// TwinCAT 3 PLC project PLC
// ProgramVersion: 3.1.4024.0
// libraries:
//   EfficientIO Communicator, * (EfficientIO)
//   EfficientIO Energy Basic, * (EfficientIO)
//   EfficientIO ModbusTCP, * (EfficientIO)
//   Lynus Persistent Data V1, * (Lynus AG)
//   Lynus Standards, * (EfficientIO)
//   Tc2_ModbusSrv, * (Beckhoff Automation GmbH)
//   Tc2_Standard, * (Beckhoff Automation GmbH)
//   Tc2_System, * (Beckhoff Automation GmbH)
//   Tc2_Utilities, * (Beckhoff Automation GmbH)
//   Tc3_Module, * (Beckhoff Automation GmbH)
// project tree:
//   / FastTask.TcTTO, MiddleTask.TcTTO, SlowTask.TcTTO
//   FB/ FB_ModBus_100Registers_FC3.TcPOU, FB_Socomec_I31.TcPOU, FB_Socomec_IO20.TcPOU, FB_Socomec_I61.TcPOU, FB_Socomec_IO10.TcPOU
//   POUs/ MAIN.TcPOU, prgE9.TcPOU, prgComEffIO.TcPOU, prgE5.TcPOU, prgRWEffIO.TcPOU, prgVarEffIO.TcPOU
// real-time tasks:
//   TASK SlowTask: cycle T#20ms, priority 21, ADS port 351
//   TASK MiddleTask: cycle T#10ms, priority 20, ADS port 352
//   TASK FastTask: cycle T#5ms, priority 19, ADS port 353

CONFIGURATION PLC
    RESOURCE PLC ON TwinCAT3
        TASK FastTask(INTERVAL := T#5ms, PRIORITY := 19);
        TASK MiddleTask(INTERVAL := T#10ms, PRIORITY := 20);
        TASK SlowTask(INTERVAL := T#20ms, PRIORITY := 21);
        PROGRAM prgRWEffIO WITH FastTask : prgRWEffIO;
        PROGRAM prgVarEffIO WITH FastTask : prgVarEffIO;
        PROGRAM MAIN WITH MiddleTask : MAIN;
        PROGRAM prgE5 WITH MiddleTask : prgE5;
        PROGRAM prgE9 WITH MiddleTask : prgE9;
        PROGRAM prgComEffIO WITH SlowTask : prgComEffIO;
    END_RESOURCE
END_CONFIGURATION

// ---- POUs/prgRWEffIO.TcPOU
PROGRAM prgRWEffIO
VAR
	fbRW1		: FB_ReadWrite_V2;
END_VAR

fbRW1(
	eUploadType:= eSelectDataUploadType.e_Change_Intervall5min, 
	bBusy=> , 
	bError=> , 
	udiErrorCodeOut=> , 
	eErrorReadWrite_Out=> );

END_PROGRAM

// ---- POUs/prgVarEffIO.TcPOU
PROGRAM prgVarEffIO
VAR
	fbVar		: FB_VarInfo_V3;
END_VAR

fbVar(
	bReadInfo:= , 
	eTMCFile:= eSelectTMCFile.eDontUseTMCFile, 
	eSavePositionTMCFile:= eSavePositionOnPLC.ePostionC, 
	udiCounterFoundVariables=> , 
	bError=> , 
	bBusy=> , 
	byProgress=> , 
	udiErrorCodeOut=> , 
	eErrorVarInfo_Out=> , 
	sVarWithError=> );

END_PROGRAM

// ---- POUs/MAIN.TcPOU
PROGRAM MAIN
VAR
	FB_Read_MB :FB_ModBus_100Registers_FC3;
	m_Enable: BOOL ;
	str_IP: STRING(15):= '192.168.8.2';
	word_Adress: WORD;
	usint_Quantity: USINT;
	byte_slaveID: BYTE;

	lr_Mischanlage_Gesamt_Freq : LREAL;		//{#lynus.ag#()}
	lr_Mischanlage_Gesamt_L1N : LREAL;		//{#lynus.ag#()}
	lr_Mischanlage_Gesamt_L2N : LREAL;		//{#lynus.ag#()}
	lr_Mischanlage_Gesamt_L3N : LREAL;		//{#lynus.ag#()}
	lr_Mischanlage_Gesamt_L1L2 : LREAL;		//{#lynus.ag#()}
	lr_Mischanlage_Gesamt_L2L3 : LREAL;		//{#lynus.ag#()}
	lr_Mischanlage_Gesamt_L3L1 : LREAL;		//{#lynus.ag#()}
	lr_Mischanlage_Gesamt_I1 : LREAL;		//{#lynus.ag#()}
	lr_Mischanlage_Gesamt_I2 : LREAL;		//{#lynus.ag#()}
	lr_Mischanlage_Gesamt_I3 : LREAL;		//{#lynus.ag#()}
	lr_Mischanlage_Gesamt_N : LREAL;		//{#lynus.ag#()}
	lr_Mischanlage_Gesamt_S : LREAL;		//{#lynus.ag#()}
	lr_Mischanlage_Gesamt_P : LREAL;		//{#lynus.ag#()}
	lr_Mischanlage_Gesamt_Q : LREAL;		//{#lynus.ag#()}
	lr_Mischanlage_Gesamt_PF : LREAL;		//{#lynus.ag#()}
	
	lr_VerteilerRC_Kalt_Freq : LREAL;		//{#lynus.ag#()}
	lr_VerteilerRC_Kalt_L1N : LREAL;		//{#lynus.ag#()}
	lr_VerteilerRC_Kalt_L2N : LREAL;		//{#lynus.ag#()}
	lr_VerteilerRC_Kalt_L3N : LREAL;		//{#lynus.ag#()}
	lr_VerteilerRC_Kalt_L1L2 : LREAL;		//{#lynus.ag#()}
	lr_VerteilerRC_Kalt_L2L3 : LREAL;		//{#lynus.ag#()}
	lr_VerteilerRC_Kalt_L3L1 : LREAL;		//{#lynus.ag#()}
	lr_VerteilerRC_Kalt_I1 : LREAL;			//{#lynus.ag#()}
	lr_VerteilerRC_Kalt_I2 : LREAL;			//{#lynus.ag#()}
	lr_VerteilerRC_Kalt_I3 : LREAL;			//{#lynus.ag#()}
	lr_VerteilerRC_Kalt_N : LREAL;			//{#lynus.ag#()}
	lr_VerteilerRC_Kalt_S : LREAL;			//{#lynus.ag#()}
	lr_VerteilerRC_Kalt_P : LREAL;			//{#lynus.ag#()}
	lr_VerteilerRC_Kalt_Q : LREAL;			//{#lynus.ag#()}
	lr_VerteilerRC_Kalt_PF : LREAL;			//{#lynus.ag#()}
	

	lr_Begleitheizung_Freq : LREAL;			//{#lynus.ag#()}
	lr_Begleitheizung_L1N : LREAL;			//{#lynus.ag#()}
	lr_Begleitheizung_L2N : LREAL;			//{#lynus.ag#()}
	lr_Begleitheizung_L3N : LREAL;			//{#lynus.ag#()}
	lr_Begleitheizung_L1L2 : LREAL;			//{#lynus.ag#()}
	lr_Begleitheizung_L2L3 : LREAL;			//{#lynus.ag#()}
	lr_Begleitheizung_L3L1 : LREAL;			//{#lynus.ag#()}
	lr_Begleitheizung_I1 : LREAL;			//{#lynus.ag#()}
	lr_Begleitheizung_I2 : LREAL;			//{#lynus.ag#()}
	lr_Begleitheizung_I3 : LREAL;			//{#lynus.ag#()}
	lr_Begleitheizung_N : LREAL;			//{#lynus.ag#()}
	lr_Begleitheizung_S : LREAL;			//{#lynus.ag#()}
	lr_Begleitheizung_P : LREAL;			//{#lynus.ag#()}
	lr_Begleitheizung_Q : LREAL;			//{#lynus.ag#()}
	lr_Begleitheizung_PF : LREAL;			//{#lynus.ag#()}

	lr_Nebenantriebe_Freq : LREAL;			//{#lynus.ag#()}
	lr_Nebenantriebe_L1N : LREAL;			//{#lynus.ag#()}
	lr_Nebenantriebe_L2N : LREAL;			//{#lynus.ag#()}
	lr_Nebenantriebe_L3N : LREAL;			//{#lynus.ag#()}
	lr_Nebenantriebe_L1L2 : LREAL;			//{#lynus.ag#()}
	lr_Nebenantriebe_L2L3 : LREAL;			//{#lynus.ag#()}
	lr_Nebenantriebe_L3L1 : LREAL;			//{#lynus.ag#()}
	lr_Nebenantriebe_I1 : LREAL;			//{#lynus.ag#()}
	lr_Nebenantriebe_I2 : LREAL;			//{#lynus.ag#()}
	lr_Nebenantriebe_I3 : LREAL;			//{#lynus.ag#()}
	lr_Nebenantriebe_N : LREAL;				//{#lynus.ag#()}
	lr_Nebenantriebe_S : LREAL;				//{#lynus.ag#()}
	lr_Nebenantriebe_P : LREAL;				//{#lynus.ag#()}
	lr_Nebenantriebe_Q : LREAL;				//{#lynus.ag#()}
	lr_Nebenantriebe_PF : LREAL;			//{#lynus.ag#()}
	
	lr_Rest_P : LREAL;								//{#lynus.ag#()}
	lr_GasmessungWTMenge_m3h 	: LREAL;			//{#lynus.ag#()}
	lr_GasmessungWTMenge_m3h_2 	: LREAL;			//{#lynus.ag#()}
	lr_GasmessungWTTemp_C 		: LREAL;			//{#lynus.ag#()}
	lr_GasmessungWTDruck_bar 	: LREAL;			//{#lynus.ag#()}
	m_Brennerstart			 	: BOOL;			//{#lynus.ag#()}
	m_Mischerstart			 	: BOOL;			//{#lynus.ag#()}
	m_Oelzaehler			 	: BOOL;			//{#lynus.ag#()}
	
	FB_Read_Socomec_I61 	: FB_Socomec_I61;
	FB_Read_Socomec_IO20	: FB_Socomec_IO20;
	FB_Read_Socomec_IO10	: FB_Socomec_IO10;
	i_State_ModbusCall: INT;				
	ton_TimeOutState: ton;
	tof_TimeOut_Active: tof;
	i_State_ModbusCall_old: INT;
	int_errorCount: INT;
	m_TimeOutActive: BOOL;					//{#lynus.ag#()}
	i_State_ErrorActive: INT;				//{#lynus.ag#()}
	lr_Rest_P_Temp: LREAL;
END_VAR


lr_Rest_P := LIMIT(	0,
					lr_Mischanlage_Gesamt_P - lr_VerteilerRC_Kalt_P - lr_Begleitheizung_P - lr_Nebenantriebe_P
						- prgE5.lr_RC_Anlage_P - prgE5.lr_RC_Trommel_P  
						- prgE9.lr_Bitumentank_4_P - prgE9.lr_Dosierpumpe_1_P - prgE9.lr_Bitumenfuellpumpe_1_P - prgE9.lr_Dosierpumpe_2_P  - prgE9.lr_Bitumentank_1_P - prgE9.lr_Bitumentank_2_P - prgE9.lr_Bitumentank_3_P
					,1000);
lr_Rest_P_Temp :=	lr_Mischanlage_Gesamt_P - lr_VerteilerRC_Kalt_P - lr_Begleitheizung_P - lr_Nebenantriebe_P
						- prgE5.lr_RC_Anlage_P - prgE5.lr_RC_Trommel_P  
						- prgE9.lr_Bitumentank_4_P - prgE9.lr_Dosierpumpe_1_P - prgE9.lr_Bitumenfuellpumpe_1_P - prgE9.lr_Dosierpumpe_2_P  - prgE9.lr_Bitumentank_1_P - prgE9.lr_Bitumentank_2_P - prgE9.lr_Bitumentank_3_P;
CASE i_State_ModbusCall OF
	0: 	// wait state
		i_State_ModbusCall := 10;
	
	10:	// first Modbus Poll Call
		FB_Read_Socomec_I61.m_Start := TRUE;
		FB_Read_Socomec_I61.byte_slaveID := 3;
		FB_Read_Socomec_I61.w_Adress := 18442;
		i_State_ModbusCall := i_State_ModbusCall + 1;
	
	11: // wait for received data
		FB_Read_Socomec_I61.m_Start := FALSE;
		IF FB_Read_Socomec_I61.iStateModbusRead = 30 THEN
			lr_Mischanlage_Gesamt_Freq	:=		FB_Read_Socomec_I61.lr_Freq_Hz	;	
			lr_Mischanlage_Gesamt_L1N	:=		FB_Read_Socomec_I61.lr_L1N_V	;	
			lr_Mischanlage_Gesamt_L2N	:=		FB_Read_Socomec_I61.lr_L2N_V	;	
			lr_Mischanlage_Gesamt_L3N	:=		FB_Read_Socomec_I61.lr_L3N_V	;	
			lr_Mischanlage_Gesamt_L1L2	:=		FB_Read_Socomec_I61.lr_L1L2_V	;	
			lr_Mischanlage_Gesamt_L2L3	:=		FB_Read_Socomec_I61.lr_L2L3_V	;	
			lr_Mischanlage_Gesamt_L3L1	:=		FB_Read_Socomec_I61.lr_L3L1_V	;	
			lr_Mischanlage_Gesamt_I1	:=		FB_Read_Socomec_I61.lr_I1_A		;	
			lr_Mischanlage_Gesamt_I2	:=		FB_Read_Socomec_I61.lr_I2_A		;	
			lr_Mischanlage_Gesamt_I3	:=		FB_Read_Socomec_I61.lr_I3_A		;	
			lr_Mischanlage_Gesamt_N		:=		FB_Read_Socomec_I61.lr_N_A		;	
			lr_Mischanlage_Gesamt_P		:=		FB_Read_Socomec_I61.lr_P_kW		;	
			lr_Mischanlage_Gesamt_Q		:=		FB_Read_Socomec_I61.lr_Q_kVAr	;	
			lr_Mischanlage_Gesamt_S		:=		FB_Read_Socomec_I61.lr_S_kVA	;	
			lr_Mischanlage_Gesamt_PF	:=		FB_Read_Socomec_I61.lr_PF		;		
			
			i_State_ModbusCall := i_State_ModbusCall +1;
		END_IF            
		IF FB_Read_Socomec_I61.iStateModbusError = 300 OR ton_TimeOutState.Q THEN
			i_State_ModbusCall := i_State_ModbusCall +1;
		END_IF
	
	12: // wait for FB_Read_Socomec_I61 to be in state 0
		IF FB_Read_Socomec_I61.iStateModbusRead = 0 OR ton_TimeOutState.Q THEN
			i_State_ModbusCall := i_State_ModbusCall + 8;
		END_IF

	20:	// next Modbus Poll Call
		FB_Read_Socomec_I61.m_Start := TRUE;
		FB_Read_Socomec_I61.byte_slaveID := 4;
		FB_Read_Socomec_I61.w_Adress := 18442;
		i_State_ModbusCall := i_State_ModbusCall + 1;
	
	21: // wait for received data
		FB_Read_Socomec_I61.m_Start := FALSE;
		IF FB_Read_Socomec_I61.iStateModbusRead = 30 THEN
			lr_VerteilerRC_Kalt_Freq	:=		FB_Read_Socomec_I61.lr_Freq_Hz	;	
			lr_VerteilerRC_Kalt_L1N		:=		FB_Read_Socomec_I61.lr_L1N_V	;	
			lr_VerteilerRC_Kalt_L2N		:=		FB_Read_Socomec_I61.lr_L2N_V	;	
			lr_VerteilerRC_Kalt_L3N		:=		FB_Read_Socomec_I61.lr_L3N_V	;	
			lr_VerteilerRC_Kalt_L1L2	:=		FB_Read_Socomec_I61.lr_L1L2_V	;	
			lr_VerteilerRC_Kalt_L2L3	:=		FB_Read_Socomec_I61.lr_L2L3_V	;	
			lr_VerteilerRC_Kalt_L3L1	:=		FB_Read_Socomec_I61.lr_L3L1_V	;	
			lr_VerteilerRC_Kalt_I1		:=		FB_Read_Socomec_I61.lr_I1_A		;	
			lr_VerteilerRC_Kalt_I2		:=		FB_Read_Socomec_I61.lr_I2_A		;	
			lr_VerteilerRC_Kalt_I3		:=		FB_Read_Socomec_I61.lr_I3_A		;	
			lr_VerteilerRC_Kalt_N		:=		FB_Read_Socomec_I61.lr_N_A		;	
			lr_VerteilerRC_Kalt_P		:=		FB_Read_Socomec_I61.lr_P_kW		;	
			lr_VerteilerRC_Kalt_Q		:=		FB_Read_Socomec_I61.lr_Q_kVAr	;	
			lr_VerteilerRC_Kalt_S		:=		FB_Read_Socomec_I61.lr_S_kVA	;	
			lr_VerteilerRC_Kalt_PF		:=		FB_Read_Socomec_I61.lr_PF		;		
			
			i_State_ModbusCall := i_State_ModbusCall +1;
		END_IF            
		IF FB_Read_Socomec_I61.iStateModbusError = 300 OR ton_TimeOutState.Q THEN
			i_State_ModbusCall := i_State_ModbusCall +1;
		END_IF
	
	22: // wait for FB_Read_Socomec_I61 to be in state 0
		IF FB_Read_Socomec_I61.iStateModbusRead = 0 OR ton_TimeOutState.Q THEN
			i_State_ModbusCall := i_State_ModbusCall + 8;
		END_IF
	
	30:	// next Modbus Poll Call
		FB_Read_Socomec_I61.m_Start := TRUE;
		FB_Read_Socomec_I61.byte_slaveID := 3;
		FB_Read_Socomec_I61.w_Adress := 20490;
		i_State_ModbusCall := i_State_ModbusCall + 1;
	
	31: // wait for received data
		FB_Read_Socomec_I61.m_Start := FALSE;
		IF FB_Read_Socomec_I61.iStateModbusRead = 30 THEN
			lr_Begleitheizung_Freq	:=		FB_Read_Socomec_I61.lr_Freq_Hz	;	
			lr_Begleitheizung_L1N	:=		FB_Read_Socomec_I61.lr_L1N_V	;	
			lr_Begleitheizung_L2N	:=		FB_Read_Socomec_I61.lr_L2N_V	;	
			lr_Begleitheizung_L3N	:=		FB_Read_Socomec_I61.lr_L3N_V	;	
			lr_Begleitheizung_L1L2	:=		FB_Read_Socomec_I61.lr_L1L2_V	;	
			lr_Begleitheizung_L2L3	:=		FB_Read_Socomec_I61.lr_L2L3_V	;	
			lr_Begleitheizung_L3L1	:=		FB_Read_Socomec_I61.lr_L3L1_V	;	
			lr_Begleitheizung_I1	:=		FB_Read_Socomec_I61.lr_I1_A		;	
			lr_Begleitheizung_I2	:=		FB_Read_Socomec_I61.lr_I2_A		;	
			lr_Begleitheizung_I3	:=		FB_Read_Socomec_I61.lr_I3_A		;	
			lr_Begleitheizung_N		:=		FB_Read_Socomec_I61.lr_N_A		;	
			lr_Begleitheizung_P		:=		FB_Read_Socomec_I61.lr_P_kW		;	
			lr_Begleitheizung_Q		:=		FB_Read_Socomec_I61.lr_Q_kVAr	;	
			lr_Begleitheizung_S		:=		FB_Read_Socomec_I61.lr_S_kVA	;	
			lr_Begleitheizung_PF	:=		FB_Read_Socomec_I61.lr_PF		;		
			
			i_State_ModbusCall := i_State_ModbusCall +1;
		END_IF            
		IF FB_Read_Socomec_I61.iStateModbusError = 300 OR ton_TimeOutState.Q THEN
			i_State_ModbusCall := i_State_ModbusCall +1;
		END_IF
	
	32: // wait for FB_Read_Socomec_I61 to be in state 0
		IF FB_Read_Socomec_I61.iStateModbusRead = 0 OR ton_TimeOutState.Q THEN
			i_State_ModbusCall := i_State_ModbusCall + 8;
		END_IF
	
	40:	// next Modbus Poll Call
		FB_Read_Socomec_I61.m_Start := TRUE;
		FB_Read_Socomec_I61.byte_slaveID := 4;
		FB_Read_Socomec_I61.w_Adress := 20490;
		i_State_ModbusCall := i_State_ModbusCall + 1;
	
	41: // wait for received data
		FB_Read_Socomec_I61.m_Start := FALSE;
		IF FB_Read_Socomec_I61.iStateModbusRead = 30 THEN
			lr_Nebenantriebe_Freq	:=		FB_Read_Socomec_I61.lr_Freq_Hz	;	
			lr_Nebenantriebe_L1N	:=		FB_Read_Socomec_I61.lr_L1N_V	;	
			lr_Nebenantriebe_L2N	:=		FB_Read_Socomec_I61.lr_L2N_V	;	
			lr_Nebenantriebe_L3N	:=		FB_Read_Socomec_I61.lr_L3N_V	;	
			lr_Nebenantriebe_L1L2	:=		FB_Read_Socomec_I61.lr_L1L2_V	;	
			lr_Nebenantriebe_L2L3	:=		FB_Read_Socomec_I61.lr_L2L3_V	;	
			lr_Nebenantriebe_L3L1	:=		FB_Read_Socomec_I61.lr_L3L1_V	;	
			lr_Nebenantriebe_I1		:=		FB_Read_Socomec_I61.lr_I1_A		;	
			lr_Nebenantriebe_I2		:=		FB_Read_Socomec_I61.lr_I2_A		;	
			lr_Nebenantriebe_I3		:=		FB_Read_Socomec_I61.lr_I3_A		;	
			lr_Nebenantriebe_N		:=		FB_Read_Socomec_I61.lr_N_A		;	
			lr_Nebenantriebe_P		:=		FB_Read_Socomec_I61.lr_P_kW		;	
			lr_Nebenantriebe_Q		:=		FB_Read_Socomec_I61.lr_Q_kVAr	;	
			lr_Nebenantriebe_S		:=		FB_Read_Socomec_I61.lr_S_kVA	;	
			lr_Nebenantriebe_PF		:=		FB_Read_Socomec_I61.lr_PF		;		
			
			i_State_ModbusCall := i_State_ModbusCall +1;
		END_IF            
		IF FB_Read_Socomec_I61.iStateModbusError = 300 OR ton_TimeOutState.Q THEN
			i_State_ModbusCall := i_State_ModbusCall +1;
		END_IF
	
	42: // wait for FB_Read_Socomec_I61 to be in state 0
		IF FB_Read_Socomec_I61.iStateModbusRead = 0 OR ton_TimeOutState.Q THEN
			i_State_ModbusCall := i_State_ModbusCall + 8;
		END_IF


	50:	// next Modbus Poll Call		first IO20 call
		FB_Read_Socomec_IO20.m_Start := TRUE;
		FB_Read_Socomec_IO20.byte_slaveID := 5;
		FB_Read_Socomec_IO20.w_Adress := 11589;
		i_State_ModbusCall := i_State_ModbusCall + 1;
	
	51: // wait for received data
		FB_Read_Socomec_IO20.m_Start := FALSE;
		IF FB_Read_Socomec_IO20.iStateModbusRead = 30 THEN
			lr_GasmessungWTMenge_m3h := LIMIT(0,2150.0/16.0*(FB_Read_Socomec_IO20.lr_Value_mA-4),2150);		// 4-20mA = 0-2150 m3/h
			lr_GasmessungWTMenge_m3h_2 := LIMIT(0,FB_Read_Socomec_IO20.lr_Value_mA,2150);					// plain Output Socomec
			i_State_ModbusCall := i_State_ModbusCall +1;
		END_IF            
		IF FB_Read_Socomec_I61.iStateModbusError = 300 OR ton_TimeOutState.Q THEN
			i_State_ModbusCall := i_State_ModbusCall +1;
		END_IF
	
	52: // wait for FB_Read_Socomec_IO20 to be in state 0
		IF FB_Read_Socomec_IO20.iStateModbusRead = 0 OR ton_TimeOutState.Q THEN
			i_State_ModbusCall := i_State_ModbusCall + 8;
		END_IF
		
	60:	// next Modbus Poll Call		second IO20 call
		FB_Read_Socomec_IO20.m_Start := TRUE;
		FB_Read_Socomec_IO20.byte_slaveID := 5;
		FB_Read_Socomec_IO20.w_Adress := 11621;
		i_State_ModbusCall := i_State_ModbusCall + 1;
	
	61: // wait for received data
		FB_Read_Socomec_IO20.m_Start := FALSE;
		IF FB_Read_Socomec_IO20.iStateModbusRead = 30 THEN
			lr_GasmessungWTTemp_C := LIMIT(-20,100.0/16.0*(FB_Read_Socomec_IO20.lr_Value_mA-4)-20,80);		// 4-20mA = -20-80 °C
				
			i_State_ModbusCall := i_State_ModbusCall +1;
		END_IF            
		IF FB_Read_Socomec_IO20.iStateModbusError = 300 OR ton_TimeOutState.Q THEN
			i_State_ModbusCall := i_State_ModbusCall +1;
		END_IF
	
	62: // wait for FB_Read_Socomec_IO20 to be in state 0
		IF FB_Read_Socomec_IO20.iStateModbusRead = 0 OR ton_TimeOutState.Q THEN
			i_State_ModbusCall := i_State_ModbusCall + 8;
		END_IF
	70:	// next Modbus Poll Call		third IO20 call
		FB_Read_Socomec_IO20.m_Start := TRUE;
		FB_Read_Socomec_IO20.byte_slaveID := 6;
		FB_Read_Socomec_IO20.w_Adress := 11589;
		i_State_ModbusCall := i_State_ModbusCall + 1;
	
	71: // wait for received data
		FB_Read_Socomec_IO20.m_Start := FALSE;
		IF FB_Read_Socomec_IO20.iStateModbusRead = 30 THEN
			lr_GasmessungWTDruck_bar :=	LIMIT(0,(5.0/16.0) * (FB_Read_Socomec_IO20.lr_Value_mA-4),5);		// 4-20mA = 0-5 bar
			i_State_ModbusCall := i_State_ModbusCall +1;
		END_IF            
		IF FB_Read_Socomec_IO20.iStateModbusError = 300 OR ton_TimeOutState.Q THEN
			i_State_ModbusCall := i_State_ModbusCall +1;
		END_IF
	
	72: // wait for FB_Read_Socomec_IO20 to be in state 0
		IF FB_Read_Socomec_IO20.iStateModbusRead = 0 OR ton_TimeOutState.Q THEN
			i_State_ModbusCall := i_State_ModbusCall + 8;
		END_IF

	80:	// next Modbus Poll Call		first IO20 call
		FB_Read_Socomec_IO10.m_Start := TRUE;
		FB_Read_Socomec_IO10.byte_slaveID := 7;
		FB_Read_Socomec_IO10.w_Adress := 11520;
		i_State_ModbusCall := i_State_ModbusCall + 1;
	
	81: // wait for received data
		FB_Read_Socomec_IO10.m_Start := FALSE;
		IF FB_Read_Socomec_IO10.iStateModbusRead = 30 THEN
			m_Brennerstart := FB_Read_Socomec_IO10.m_Input_Active;		
				
			i_State_ModbusCall := i_State_ModbusCall +1;
		END_IF            
		IF FB_Read_Socomec_IO10.iStateModbusError = 300 OR ton_TimeOutState.Q THEN
			i_State_ModbusCall := i_State_ModbusCall +1;
		END_IF
	
	82: // wait for FB_Read_Socomec_IO10 to be in state 0
		IF FB_Read_Socomec_IO10.iStateModbusRead = 0 OR ton_TimeOutState.Q THEN
			i_State_ModbusCall := i_State_ModbusCall + 8;
		END_IF

	90:	// next Modbus Poll Call		first IO20 call
		FB_Read_Socomec_IO10.m_Start := TRUE;
		FB_Read_Socomec_IO10.byte_slaveID := 7;
		FB_Read_Socomec_IO10.w_Adress := 11522;
		i_State_ModbusCall := i_State_ModbusCall + 1;
	
	91: // wait for received data
		FB_Read_Socomec_IO10.m_Start := FALSE;
		IF FB_Read_Socomec_IO10.iStateModbusRead = 30 THEN
			m_Mischerstart := FB_Read_Socomec_IO10.m_Input_Active;		
				
			i_State_ModbusCall := i_State_ModbusCall +1;
		END_IF            
		IF FB_Read_Socomec_IO10.iStateModbusError = 300 OR ton_TimeOutState.Q THEN
			i_State_ModbusCall := i_State_ModbusCall +1;
		END_IF
	
	92: // wait for FB_Read_Socomec_IO10 to be in state 0
		IF FB_Read_Socomec_IO10.iStateModbusRead = 0 OR ton_TimeOutState.Q THEN
			i_State_ModbusCall := i_State_ModbusCall + 8;
		END_IF
	100:	// next Modbus Poll Call		first IO20 call
		FB_Read_Socomec_IO10.m_Start := TRUE;
		FB_Read_Socomec_IO10.byte_slaveID := 7;
		FB_Read_Socomec_IO10.w_Adress := 11524;
		i_State_ModbusCall := i_State_ModbusCall + 1;
	
	101: // wait for received data
		FB_Read_Socomec_IO10.m_Start := FALSE;
		IF FB_Read_Socomec_IO10.iStateModbusRead = 30 THEN
			m_Oelzaehler := FB_Read_Socomec_IO10.m_Input_Active;		
				
			i_State_ModbusCall := i_State_ModbusCall +1;
		END_IF            
		IF FB_Read_Socomec_IO10.iStateModbusError = 300 OR ton_TimeOutState.Q THEN
			i_State_ModbusCall := i_State_ModbusCall +1;
		END_IF
	
	102: // wait for FB_Read_Socomec_IO10 to be in state 0
		IF FB_Read_Socomec_IO10.iStateModbusRead = 0 OR ton_TimeOutState.Q THEN
			i_State_ModbusCall := i_State_ModbusCall + 8;
		END_IF				
		
	110: 
		i_State_ModbusCall := 0;
END_CASE

ton_TimeOutState(	IN:= i_State_ModbusCall = i_State_ModbusCall_old, 
					PT:= T#30S, 
					Q=> , 
					ET=> );

i_State_ModbusCall_old := i_State_ModbusCall; 

IF ton_TimeOutState.Q THEN
//	i_State_ModbusCall := 0;
	int_errorCount := int_errorCount  + 1; 
END_IF


tof_TimeOut_Active(	IN:= ton_TimeOutState.Q, 
					PT:=	T#5S , 
					Q=> m_TimeOutActive, 
					ET=> );
IF tof_TimeOut_Active.Q THEN
	 i_State_ErrorActive := i_State_ModbusCall; 
END_IF


FB_Read_Socomec_I61(
	m_Start:= , 
	str_IPAdress:= str_IP , 
	w_Adress:= , 
	uint_port:= , 
	byte_slaveID:= , 
	m_PollSuccessful=> , 
	lr_Freq_Hz=> , 
	lr_L1N_V=> , 
	lr_L2N_V=> , 
	lr_L3N_V=> , 
	lr_L1L2_V=> , 
	lr_L2L3_V=> , 
	lr_L3L1_V=> , 
	lr_I1_A=> , 
	lr_I2_A=> , 
	lr_I3_A=> , 
	lr_N_A=> , 
	lr_P_kW=> , 
	lr_Q_kVAr=> , 
	lr_S_kVA=> , 
	lr_PF=> , 
	udint_Error_ID=> );

FB_Read_Socomec_IO20(
	m_Start:= , 
	str_IPAdress:= str_IP, 
	w_Adress:= , 
	uint_port:= , 
	byte_slaveID:= , 
	m_PollSuccessful=> , 
	lr_Value_mA=> , 
	udint_Error_ID=> );

FB_Read_Socomec_IO10(
	m_Start:= , 
	str_IPAdress:= str_IP , 
	w_Adress:= , 
	uint_port:= , 
	byte_slaveID:= , 
	m_PollSuccessful=> , 
	m_Input_Active=> , 
	udint_Error_ID=> );	


FB_Read_MB(
	m_Enable:= m_Enable, 
	str_IPAdress:= str_IP,
	w_Adress:= word_Adress, 
	usint_Quantity:= usint_Quantity, 
	byte_slaveID:=byte_slaveID,
	uint_port := ,
	m_PollSuccessful=> , 
	w_Array_Received=> , 
	udint_Error_ID=> );

END_PROGRAM

// ---- FB/FB_ModBus_100Registers_FC3.TcPOU
FUNCTION_BLOCK FB_ModBus_100Registers_FC3
VAR_INPUT PERSISTENT
	m_Enable					: BOOL;						//Enable the Fuctionblock and his logic
	str_IPAdress				: STRING(15);				//IP Adress of the meter
	w_Adress					: WORD;						//modbus adress
	usint_Quantity				: USINT;					//Number of Words to get polled, max 100
	uint_port					: UINT:=502;				//ModbusPort
	byte_slaveID				: BYTE;						//SlaveID of the meter
END_VAR
VAR_OUTPUT
	m_PollSuccessful			: BOOL;						//Poll succesfull		
	w_Array_Received			: ARRAY[1..100] OF WORD;	// received data
	udint_Error_ID				: UDINT;					// ERR ID FB_MBReadRegs
END_VAR
VAR
	
	timer_Delay					: TON;						//Timer for Delay between Requests
	
	timer_DelayStart			: TON;						//Timer to start the state machine with Delay after enabling or after the system ist restartet
	
	timer_TimeOut				: TON;						//Timer for Timeout MB Read
	
	iStateModbusRead			: INT;						//State machine for read out Data over Modbus RTU
	
	fbMBRead_FC3				: FB_MBReadRegs  ;		//Modbus Read Function (FC3)
	
	ftrig_PEnable				: f_trig;					//Internal positive Edge
	
	iStateModbusError			: INT;						//State machine for error out Data over Modbus TCP/IP	
	
	FPError_FC_3				: R_TRIG;					//Internal positive Edge
	
	arrBuffer_FC3				: ARRAY[1..100] OF WORD;		//Buffer with Data from FC3
	
	timer_Connection_ok			: TON;
	int_Data_Received			: INT;
	
	m_MBTCPError				: BOOL;
	
	int_Data_Received_old		: INT;
	
	timer_Connection_ok_TOF	: TOF;
	
	fbConvertWordToDword		: FB_CV_WORD_TO_DWORD;			//Convert Word to Dword
	
	m_Poll_ok: BOOL;
	
	timer_Wait: Ton;
	int_TimeoutError: INT;
	int_FC3Error: INT;

END_VAR

(*	{attribute 'hide'}--------------------------------------------------------------------------------------------Limits-------------------------------------------------------------------------------------*)

w_Adress := LIMIT(0,w_Adress,60000);
usint_Quantity := LIMIT(1,usint_Quantity,100);
	
(*--------------------------------------------------------------------------------------------State Machine Read--------------------------------------------------------------------------------------*)

//Timer for Delay
timer_Delay(IN:= , PT:= T#50MS, Q=> , ET=> );

//Timeout Timer is dissabled when the Init Step is aktiv or the function is not enabled
IF iStateModbusRead = 0 OR NOT m_Enable THEN 
	timer_Timeout.IN := FALSE; 
END_IF
timer_Timeout(IN:= , PT:= T#1S, Q=> , ET=> );

//Enable with Delay that not all sockets have to be created at the same time
timer_DelayStart(IN:= m_Enable, PT:= T#1S, Q=> , ET=> );
ftrig_PEnable(CLK:= timer_DelayStart.Q, Q=> );

IF ftrig_PEnable.Q AND iStateModbusRead = 0 THEN 
	iStateModbusRead := 1; 
END_IF		
		
//Not Enabled
IF NOT m_Enable THEN 
	iStateModbusRead := 0; 
	iStateModbusError := 0; 
END_IF		
		
CASE iStateModbusRead OF

	0://Init Step 
		timer_Delay.IN := FALSE;
		fbMBRead_FC3.bExecute := FALSE;
		m_Poll_ok:=FALSE;
		int_Data_Received:=0;
	
		iStateModbusRead := 1;
	
	1://read the required registers
		//Start Read
		fbMBRead_FC3.nQuantity := usint_Quantity;
		fbMBRead_FC3.nMBAddr := w_Adress;
		fbMBRead_FC3.bExecute := TRUE;
		fbMBRead_FC3.nUnitID := byte_slaveID;
		timer_Timeout.IN := TRUE;
		IF fbMBRead_FC3.bBusy THEN 
			timer_Delay.IN := TRUE; 
		END_IF
		
		//Wait for Delay, copy Data and then next step
		IF NOT fbMBRead_FC3.bBusy AND NOT fbMBRead_FC3.bError AND timer_Delay.Q THEN
			m_Poll_ok:=TRUE;
			int_Data_Received:=int_Data_Received+1;
			m_MBTCPError := FALSE; 
			
			w_Array_Received := arrBuffer_FC3;
			
			
			//Go to Next Step
			timer_Timeout.IN := FALSE;
			fbMBRead_FC3.bExecute := FALSE;
			timer_Delay.IN := FALSE;		
			iStateModbusRead := 3;
		END_IF	

		//Error or Timeout
		IF FPError_FC_3.Q THEN 
			iStateModbusError := 300;
			int_FC3Error := int_FC3Error+1;
		ELSIF timer_Timeout.Q THEN  
			timer_Timeout.IN := FALSE; 	
			iStateModbusError := 300;
			int_TimeoutError := int_TimeoutError+1;
		END_IF
		
	
	3://Wait and go to step 1
		//1 because 0 is the Init Step for Read
		timer_Wait.IN := TRUE;
		
		IF timer_Wait.Q = TRUE THEN
			iStateModbusRead := 1;
			timer_Wait.IN :=FALSE;
		END_IF

			
		
		//Error on Master, changes on Inputs or Timeout
		IF timer_Timeout.Q THEN 
			iStateModbusError := 300; 
		END_IF
	
END_CASE

(* wait timer*)

timer_Wait(PT:=T#3S);


(*------------------------------------------------------------------Error and Warning----------------------------------------------------------------------------*)	
 
timer_Connection_ok			(In:=int_Data_Received<>int_Data_Received_old,PT:=T#10S);
timer_Connection_ok_TOF		(In:=NOT(int_Data_Received<>int_Data_Received_old) AND int_Data_Received>3 ,PT:=T#20S);
int_Data_Received_old:=int_Data_Received;
m_PollSuccessful:=NOT timer_Connection_ok.Q AND timer_Connection_ok_TOF.Q ;

(*------------------------------------------------------------------------------------------Modbus TCP Functions---------------------------------------------------------------------------------------------*)

fbMBRead_FC3(	sIPAddr:= str_IPAdress, 
				nTCPPort:= uint_port,
				cbLength:= SIZEOF(arrBuffer_FC3), 
				pDestAddr:= ADR(arrBuffer_FC3), 
				tTimeout:= T#10S,
				nErrId => udint_Error_ID);

FPError_FC_3(CLK:= fbMBRead_FC3.bError, Q=> );		

(*------------------------------------------------------------------------------------------State Machine Error---------------------------------------------------------------------------------------------*)	

CASE iStateModbusError OF
	
	300://Error
		timer_Wait.IN :=TRUE;
		timer_Delay.IN := FALSE;
		fbMBRead_FC3.bExecute := FALSE;
		m_MBTCPError := TRUE; 		
		m_Poll_ok:=FALSE;
		int_Data_Received:=0;
				//Restart from new with the Read out part after an Error
		IF timer_Wait.Q = TRUE THEN
			iStateModbusRead := 0;	
			iStateModbusError := 0;
			timer_Wait.IN :=FALSE;
			timer_Timeout.IN := FALSE;
		END_IF		
							
END_CASE

END_FUNCTION_BLOCK

// ---- FB/FB_Socomec_I61.TcPOU
FUNCTION_BLOCK FB_Socomec_I61
VAR_INPUT PERSISTENT
	m_Start						: BOOL;						//starts one modbus read out
	str_IPAdress				: STRING(15);				//IP Adress of the meter
	w_Adress					: WORD;						//modbus adress
	uint_port					: UINT:=502;				//ModbusPort
	byte_slaveID				: BYTE;						//SlaveID of the meter
END_VAR
VAR_OUTPUT
	m_PollSuccessful			: BOOL;						//Poll succesfull		
	lr_Freq_Hz					: LREAL;
	lr_L1N_V					: LREAL;	
	lr_L2N_V					: LREAL;	
	lr_L3N_V					: LREAL;	
	lr_L1L2_V					: LREAL;	
	lr_L2L3_V					: LREAL;	
	lr_L3L1_V					: LREAL;	
	lr_I1_A						: LREAL;	
	lr_I2_A						: LREAL;	
	lr_I3_A						: LREAL;	
	lr_N_A						: LREAL;	
	lr_P_kW						: LREAL;
	lr_Q_kVAr					: LREAL;
	lr_S_kVA					: LREAL;
	lr_PF						: LREAL;	
	udint_Error_ID				: UDINT;					// ERR ID FB_MBReadRegs
END_VAR
VAR
	w_Array_Received			: ARRAY[1..100] OF WORD;	// received data
	timer_Delay					: TON;						//Timer for Delay between Requests
	timer_TimeOut				: TON;						//Timer for Timeout MB Read
	iStateModbusRead			: INT;						//State machine for read out Data over Modbus RTU
	fbMBRead_FC3				: FB_MBReadRegs  ;		//Modbus Read Function (FC3)
	rtrig_Start					: r_trig;					//positive edge for starting the read out
	iStateModbusError			: INT;						//State machine for error out Data over Modbus TCP/IP	
	FPError_FC_3				: R_TRIG;					//Internal positive Edge
	arrBuffer_FC3				: ARRAY[1..100] OF WORD;		//Buffer with Data from FC3
	timer_Connection_ok			: TON;
	int_Data_Received			: INT;
	m_MBTCPError				: BOOL;
	int_Data_Received_old		: INT;
	timer_Connection_ok_TOF	: TOF;
	fbConvertWordToDword		: FB_CV_WORD_TO_DWORD;			//Convert Word to Dword
	m_Poll_ok: BOOL;
	timer_Wait: Ton;
	int_TimeoutError: INT;
	int_FC3Error: INT;
	x: INT;
	i: INT;
	fbConvertWordToudint		: FB_CV_WORD_TO_UDINT;

END_VAR

(*	{attribute 'hide'}--------------------------------------------------------------------------------------------Limits-------------------------------------------------------------------------------------*)

w_Adress := LIMIT(0,w_Adress,60000);

	
(*--------------------------------------------------------------------------------------------State Machine Read--------------------------------------------------------------------------------------*)

//Timer for Delay
timer_Delay(IN:= , PT:= T#50MS, Q=> , ET=> );

//Timeout Timer is dissabled when the Init Step is aktiv or the function is not enabled
IF iStateModbusRead >1 THEN 
	timer_Timeout.IN := FALSE; 
END_IF
timer_Timeout(IN:= , PT:= T#5S, Q=> , ET=> );

//Enable with Delay that not all sockets have to be created at the same time

rtrig_Start(CLK:= m_Start, Q=> );

CASE iStateModbusRead OF

	0://Init Step 
		timer_Delay.IN := FALSE;
		fbMBRead_FC3.bExecute := FALSE;
		m_Poll_ok:=FALSE;
		int_Data_Received:=0;
		FOR i := 1 TO 100 BY 1 DO
			w_Array_Received[i] := 0;
		END_FOR
		iStateModbusRead := 1;
	1: // wait for rtrig START	
		IF rtrig_Start.Q THEN
			iStateModbusRead := 10;
		END_IF
	
	10://read the required registers
		//Start Read
		fbMBRead_FC3.nQuantity := 50;
		fbMBRead_FC3.nMBAddr := w_Adress;
		fbMBRead_FC3.bExecute := TRUE;
		fbMBRead_FC3.nUnitID := byte_slaveID;
		timer_Timeout.IN := TRUE;
		IF fbMBRead_FC3.bBusy THEN 
			timer_Delay.IN := TRUE; 
		END_IF
		
		//Wait for Delay, copy Data and then next step
		IF NOT fbMBRead_FC3.bBusy AND NOT fbMBRead_FC3.bError AND timer_Delay.Q THEN
			m_Poll_ok:=TRUE;
			int_Data_Received:=int_Data_Received+1;
			m_MBTCPError := FALSE; 
			
			w_Array_Received := arrBuffer_FC3;
			
			
			// convert reveived data
			x:=1;
			fbConvertWordToudint(	wInputValue_1:= w_Array_Received[x], 
									wInputValue_2:= w_Array_Received[x+1], 
									eByteOrderForConvert:= eByteOrder.eBigEndian , 
									udiOutputValue=> );
			lr_Freq_Hz:= UDINT_TO_REAL(fbConvertWordToudint.udiOutputValue)/1000;
			x:=3;
			fbConvertWordToudint(	wInputValue_1:= w_Array_Received[x], 
									wInputValue_2:= w_Array_Received[x+1], 
									eByteOrderForConvert:= eByteOrder.eBigEndian , 
									udiOutputValue=> );
			lr_L1N_V:= UDINT_TO_REAL(fbConvertWordToudint.udiOutputValue)/100;
			x:=5;
			fbConvertWordToudint(	wInputValue_1:= w_Array_Received[x], 
									wInputValue_2:= w_Array_Received[x+1], 
									eByteOrderForConvert:= eByteOrder.eBigEndian , 
									udiOutputValue=> );
			lr_L2N_V:= UDINT_TO_REAL(fbConvertWordToudint.udiOutputValue)/100;
			x:=7;
			fbConvertWordToudint(	wInputValue_1:= w_Array_Received[x], 
									wInputValue_2:= w_Array_Received[x+1], 
									eByteOrderForConvert:= eByteOrder.eBigEndian , 
									udiOutputValue=> );
			lr_L3N_V:= UDINT_TO_REAL(fbConvertWordToudint.udiOutputValue)/100;
			
			x:=11;
			fbConvertWordToudint(	wInputValue_1:= w_Array_Received[x], 
									wInputValue_2:= w_Array_Received[x+1], 
									eByteOrderForConvert:= eByteOrder.eBigEndian , 
									udiOutputValue=> );
			lr_L1L2_V:= UDINT_TO_REAL(fbConvertWordToudint.udiOutputValue)/100;
			x:=13;
			fbConvertWordToudint(	wInputValue_1:= w_Array_Received[x], 
									wInputValue_2:= w_Array_Received[x+1], 
									eByteOrderForConvert:= eByteOrder.eBigEndian , 
									udiOutputValue=> );
			lr_L2L3_V:= UDINT_TO_REAL(fbConvertWordToudint.udiOutputValue)/100;
			x:=15;
			fbConvertWordToudint(	wInputValue_1:= w_Array_Received[x], 
									wInputValue_2:= w_Array_Received[x+1], 
									eByteOrderForConvert:= eByteOrder.eBigEndian , 
									udiOutputValue=> );
			lr_L3L1_V:= UDINT_TO_REAL(fbConvertWordToudint.udiOutputValue)/100;
			
			
			x:=17;
			fbConvertWordToudint(	wInputValue_1:= w_Array_Received[x], 
									wInputValue_2:= w_Array_Received[x+1], 
									eByteOrderForConvert:= eByteOrder.eBigEndian , 
									udiOutputValue=> );
			lr_I1_A:= UDINT_TO_REAL(fbConvertWordToudint.udiOutputValue)/1000;
			x:=19;
			fbConvertWordToudint(	wInputValue_1:= w_Array_Received[x], 
									wInputValue_2:= w_Array_Received[x+1], 
									eByteOrderForConvert:= eByteOrder.eBigEndian , 
									udiOutputValue=> );
			lr_I2_A:= UDINT_TO_REAL(fbConvertWordToudint.udiOutputValue)/1000;
			x:=21;
			fbConvertWordToudint(	wInputValue_1:= w_Array_Received[x], 
									wInputValue_2:= w_Array_Received[x+1], 
									eByteOrderForConvert:= eByteOrder.eBigEndian , 
									udiOutputValue=> );
			lr_I3_A:= UDINT_TO_REAL(fbConvertWordToudint.udiOutputValue)/1000;
			x:=23;
			fbConvertWordToudint(	wInputValue_1:= w_Array_Received[x], 
									wInputValue_2:= w_Array_Received[x+1], 
									eByteOrderForConvert:= eByteOrder.eBigEndian , 
									udiOutputValue=> );
			lr_N_A:= UDINT_TO_REAL(fbConvertWordToudint.udiOutputValue)/1000;
			
			x:=35;
			lr_P_kW := DINT_TO_LREAL(DWORD_TO_DINT(w_Array_Received[x]*65536 + w_Array_Received[x+1]))/1000;
			
			x:=37;
			lr_Q_kVAr := DINT_TO_LREAL(DWORD_TO_DINT(w_Array_Received[x]*65536 + w_Array_Received[x+1]))/1000;
			
			
			x:=43;
			fbConvertWordToudint(	wInputValue_1:= w_Array_Received[x], 
									wInputValue_2:= w_Array_Received[x+1], 
									eByteOrderForConvert:= eByteOrder.eBigEndian , 
									udiOutputValue=> );
			lr_S_kVA:= UDINT_TO_REAL(fbConvertWordToudint.udiOutputValue)/1000;
			
			
			x:=45;
			lr_PF := (REAL_TO_LREAL(WORD_TO_INT(w_Array_Received[x])))/1000;
			
			
			//Go to Next Step
			timer_Timeout.IN := FALSE;
			fbMBRead_FC3.bExecute := FALSE;
			timer_Delay.IN := FALSE;		
			iStateModbusRead := 30;
		END_IF	

		//Error or Timeout
		IF FPError_FC_3.Q THEN 
			iStateModbusError := 300;
			int_FC3Error := int_FC3Error+1;
		ELSIF timer_Timeout.Q THEN  
			timer_Timeout.IN := FALSE; 	
			iStateModbusError := 300;
			int_TimeoutError := int_TimeoutError+1;
		END_IF
		
	
	30://Wait and go to step 1
		//1 because 0 is the Init Step for Read
		timer_Wait.IN := TRUE;
		
		IF timer_Wait.Q = TRUE THEN
			iStateModbusRead := 0;
			timer_Wait.IN :=FALSE;
		END_IF

			
		
		//Error on Master, changes on Inputs or Timeout
		IF timer_Timeout.Q THEN 
			iStateModbusError := 300; 
		END_IF
	
END_CASE

(* wait timer*)

timer_Wait(PT:=T#1S);


(*------------------------------------------------------------------Error and Warning----------------------------------------------------------------------------*)	
 
timer_Connection_ok			(In:=int_Data_Received<>int_Data_Received_old,PT:=T#10S);
timer_Connection_ok_TOF		(In:=NOT(int_Data_Received<>int_Data_Received_old) AND int_Data_Received>3 ,PT:=T#20S);
int_Data_Received_old:=int_Data_Received;
m_PollSuccessful:=NOT timer_Connection_ok.Q AND timer_Connection_ok_TOF.Q ;

(*------------------------------------------------------------------------------------------Modbus TCP Functions---------------------------------------------------------------------------------------------*)

fbMBRead_FC3(	sIPAddr:= str_IPAdress, 
				nTCPPort:= uint_port,
				cbLength:= SIZEOF(arrBuffer_FC3), 
				pDestAddr:= ADR(arrBuffer_FC3), 
				tTimeout:= T#10S,
				nErrId => udint_Error_ID);

FPError_FC_3(CLK:= fbMBRead_FC3.bError, Q=> );		

(*------------------------------------------------------------------------------------------State Machine Error---------------------------------------------------------------------------------------------*)	

CASE iStateModbusError OF
	
	300://Error
		timer_Wait.IN :=TRUE;
		timer_Delay.IN := FALSE;
		fbMBRead_FC3.bExecute := FALSE;
		m_MBTCPError := TRUE; 		
		m_Poll_ok:=FALSE;
		int_Data_Received:=0;
				//Restart from new with the Read out part after an Error
		IF timer_Wait.Q = TRUE THEN
			iStateModbusRead := 0;	
			iStateModbusError := 0;
			timer_Wait.IN :=FALSE;
			timer_Timeout.IN := FALSE;
		END_IF		
							
END_CASE

END_FUNCTION_BLOCK

// ---- FB/FB_Socomec_IO20.TcPOU
FUNCTION_BLOCK FB_Socomec_IO20
VAR_INPUT PERSISTENT
	m_Start						: BOOL;						//starts one modbus read out
	str_IPAdress				: STRING(15);				//IP Adress of the meter
	w_Adress					: WORD;						//modbus adress
	uint_port					: UINT:=502;				//ModbusPort
	byte_slaveID				: BYTE;						//SlaveID of the meter
END_VAR
VAR_OUTPUT
	m_PollSuccessful			: BOOL;						//Poll succesfull		
	lr_Value_mA					: LREAL;
	udint_Error_ID				: UDINT;					// ERR ID FB_MBReadRegs
END_VAR
VAR
	w_Array_Received			: ARRAY[1..100] OF WORD;	// received data
	timer_Delay					: TON;						//Timer for Delay between Requests
	timer_TimeOut				: TON;						//Timer for Timeout MB Read
	iStateModbusRead			: INT;						//State machine for read out Data over Modbus RTU
	fbMBRead_FC3				: FB_MBReadRegs  ;		//Modbus Read Function (FC3)
	rtrig_Start					: r_trig;					//positive edge for starting the read out
	iStateModbusError			: INT;						//State machine for error out Data over Modbus TCP/IP	
	FPError_FC_3				: R_TRIG;					//Internal positive Edge
	arrBuffer_FC3				: ARRAY[1..100] OF WORD;		//Buffer with Data from FC3
	timer_Connection_ok			: TON;
	int_Data_Received			: INT;
	m_MBTCPError				: BOOL;
	int_Data_Received_old		: INT;
	timer_Connection_ok_TOF	: TOF;
	fbConvertWordToDword		: FB_CV_WORD_TO_DWORD;			//Convert Word to Dword
	m_Poll_ok: BOOL;
	timer_Wait: Ton;
	int_TimeoutError: INT;
	int_FC3Error: INT;

	i: INT;
	fbConvertWordToudint		: FB_CV_WORD_TO_UDINT;

END_VAR

(*	{attribute 'hide'}--------------------------------------------------------------------------------------------Limits-------------------------------------------------------------------------------------*)

w_Adress := LIMIT(0,w_Adress,60000);

	
(*--------------------------------------------------------------------------------------------State Machine Read--------------------------------------------------------------------------------------*)

//Timer for Delay
timer_Delay(IN:= , PT:= T#50MS, Q=> , ET=> );

//Timeout Timer is dissabled when the Init Step is aktiv or the function is not enabled
IF iStateModbusRead >1 THEN 
	timer_Timeout.IN := FALSE; 
END_IF
timer_Timeout(IN:= , PT:= T#5S, Q=> , ET=> );

//Enable with Delay that not all sockets have to be created at the same time

rtrig_Start(CLK:= m_Start, Q=> );

CASE iStateModbusRead OF

	0://Init Step 
		timer_Delay.IN := FALSE;
		fbMBRead_FC3.bExecute := FALSE;
		m_Poll_ok:=FALSE;
		int_Data_Received:=0;
		FOR i := 1 TO 100 BY 1 DO
			w_Array_Received[i] := 0;
		END_FOR
		iStateModbusRead := 1;
	1: // wait for rtrig START	
		IF rtrig_Start.Q THEN
			iStateModbusRead := 10;
		END_IF
	
	10://read the required registers
		//Start Read
		fbMBRead_FC3.nQuantity := 2;
		fbMBRead_FC3.nMBAddr := w_Adress;
		fbMBRead_FC3.bExecute := TRUE;
		fbMBRead_FC3.nUnitID := byte_slaveID;
		timer_Timeout.IN := TRUE;
		IF fbMBRead_FC3.bBusy THEN 
			timer_Delay.IN := TRUE; 
		END_IF
		
		//Wait for Delay, copy Data and then next step
		IF NOT fbMBRead_FC3.bBusy AND NOT fbMBRead_FC3.bError AND timer_Delay.Q THEN
			m_Poll_ok:=TRUE;
			int_Data_Received:=int_Data_Received+1;
			m_MBTCPError := FALSE; 
			
			w_Array_Received := arrBuffer_FC3;
			
			
			// convert reveived data
		
			fbConvertWordToudint(	wInputValue_1:= w_Array_Received[1], 
									wInputValue_2:= w_Array_Received[2], 
									eByteOrderForConvert:= eByteOrder.eBigEndian , 
									udiOutputValue=> );
		
			lr_Value_mA := UDINT_TO_REAL(fbConvertWordToudint.udiOutputValue)/1000;
			
			//Go to Next Step
			timer_Timeout.IN := FALSE;
			fbMBRead_FC3.bExecute := FALSE;
			timer_Delay.IN := FALSE;		
			iStateModbusRead := 30;
		END_IF	

		//Error or Timeout
		IF FPError_FC_3.Q THEN 
			iStateModbusError := 300;
			int_FC3Error := int_FC3Error+1;
		ELSIF timer_Timeout.Q THEN  
			timer_Timeout.IN := FALSE; 	
			iStateModbusError := 300;
			int_TimeoutError := int_TimeoutError+1;
		END_IF
		
	
	30://Wait and go to step 1
		//1 because 0 is the Init Step for Read
		timer_Wait.IN := TRUE;
		
		IF timer_Wait.Q = TRUE THEN
			iStateModbusRead := 0;
			timer_Wait.IN :=FALSE;
		END_IF

			
		
		//Error on Master, changes on Inputs or Timeout
		IF timer_Timeout.Q THEN 
			iStateModbusError := 300; 
		END_IF
	
END_CASE

(* wait timer*)

timer_Wait(PT:=T#1S);


(*------------------------------------------------------------------Error and Warning----------------------------------------------------------------------------*)	
 
timer_Connection_ok			(In:=int_Data_Received<>int_Data_Received_old,PT:=T#10S);
timer_Connection_ok_TOF		(In:=NOT(int_Data_Received<>int_Data_Received_old) AND int_Data_Received>3 ,PT:=T#20S);
int_Data_Received_old:=int_Data_Received;
m_PollSuccessful:=NOT timer_Connection_ok.Q AND timer_Connection_ok_TOF.Q ;

(*------------------------------------------------------------------------------------------Modbus TCP Functions---------------------------------------------------------------------------------------------*)

fbMBRead_FC3(	sIPAddr:= str_IPAdress, 
				nTCPPort:= uint_port,
				cbLength:= SIZEOF(arrBuffer_FC3), 
				pDestAddr:= ADR(arrBuffer_FC3), 
				tTimeout:= T#10S,
				nErrId => udint_Error_ID);

FPError_FC_3(CLK:= fbMBRead_FC3.bError, Q=> );		

(*------------------------------------------------------------------------------------------State Machine Error---------------------------------------------------------------------------------------------*)	

CASE iStateModbusError OF
	
	300://Error
		timer_Wait.IN :=TRUE;
		timer_Delay.IN := FALSE;
		fbMBRead_FC3.bExecute := FALSE;
		m_MBTCPError := TRUE; 		
		m_Poll_ok:=FALSE;
		int_Data_Received:=0;
				//Restart from new with the Read out part after an Error
		IF timer_Wait.Q = TRUE THEN
			iStateModbusRead := 0;	
			iStateModbusError := 0;
			timer_Wait.IN :=FALSE;
			timer_Timeout.IN := FALSE;
		END_IF		
							
END_CASE

END_FUNCTION_BLOCK

// ---- FB/FB_Socomec_IO10.TcPOU
FUNCTION_BLOCK FB_Socomec_IO10
VAR_INPUT PERSISTENT
	m_Start						: BOOL;						//starts one modbus read out
	str_IPAdress				: STRING(15);				//IP Adress of the meter
	w_Adress					: WORD;						//modbus adress
	uint_port					: UINT:=502;				//ModbusPort
	byte_slaveID				: BYTE;						//SlaveID of the meter
END_VAR
VAR_OUTPUT
	m_PollSuccessful			: BOOL;						//Poll succesfull		
	m_Input_Active				: BOOL;
	udint_Error_ID				: UDINT;					// ERR ID FB_MBReadRegs
END_VAR
VAR
	w_Array_Received			: ARRAY[1..100] OF WORD;	// received data
	timer_Delay					: TON;						//Timer for Delay between Requests
	timer_TimeOut				: TON;						//Timer for Timeout MB Read
	iStateModbusRead			: INT;						//State machine for read out Data over Modbus RTU
	fbMBRead_FC3				: FB_MBReadRegs  ;		//Modbus Read Function (FC3)
	rtrig_Start					: r_trig;					//positive edge for starting the read out
	iStateModbusError			: INT;						//State machine for error out Data over Modbus TCP/IP	
	FPError_FC_3				: R_TRIG;					//Internal positive Edge
	arrBuffer_FC3				: ARRAY[1..100] OF WORD;		//Buffer with Data from FC3
	timer_Connection_ok			: TON;
	int_Data_Received			: INT;
	m_MBTCPError				: BOOL;
	int_Data_Received_old		: INT;
	timer_Connection_ok_TOF	: TOF;
	m_Poll_ok: BOOL;
	timer_Wait: Ton;
	int_TimeoutError: INT;
	int_FC3Error: INT;

	i: INT;

END_VAR

(*	{attribute 'hide'}--------------------------------------------------------------------------------------------Limits-------------------------------------------------------------------------------------*)

w_Adress := LIMIT(0,w_Adress,60000);

	
(*--------------------------------------------------------------------------------------------State Machine Read--------------------------------------------------------------------------------------*)

//Timer for Delay
timer_Delay(IN:= , PT:= T#50MS, Q=> , ET=> );

//Timeout Timer is dissabled when the Init Step is aktiv or the function is not enabled
IF iStateModbusRead >1 THEN 
	timer_Timeout.IN := FALSE; 
END_IF
timer_Timeout(IN:= , PT:= T#5S, Q=> , ET=> );

//Enable with Delay that not all sockets have to be created at the same time

rtrig_Start(CLK:= m_Start, Q=> );

CASE iStateModbusRead OF

	0://Init Step 
		timer_Delay.IN := FALSE;
		fbMBRead_FC3.bExecute := FALSE;
		m_Poll_ok:=FALSE;
		int_Data_Received:=0;
		FOR i := 1 TO 100 BY 1 DO
			w_Array_Received[i] := 0;
		END_FOR
		iStateModbusRead := 1;
	1: // wait for rtrig START	
		IF rtrig_Start.Q THEN
			iStateModbusRead := 10;
		END_IF
	
	10://read the required registers
		//Start Read
		fbMBRead_FC3.nQuantity := 2;
		fbMBRead_FC3.nMBAddr := w_Adress;
		fbMBRead_FC3.bExecute := TRUE;
		fbMBRead_FC3.nUnitID := byte_slaveID;
		timer_Timeout.IN := TRUE;
		IF fbMBRead_FC3.bBusy THEN 
			timer_Delay.IN := TRUE; 
		END_IF
		
		//Wait for Delay, copy Data and then next step
		IF NOT fbMBRead_FC3.bBusy AND NOT fbMBRead_FC3.bError AND timer_Delay.Q THEN
			m_Poll_ok:=TRUE;
			int_Data_Received:=int_Data_Received+1;
			m_MBTCPError := FALSE; 
			
			w_Array_Received := arrBuffer_FC3;
			
			
			// convert reveived data
		
		
			m_Input_Active := w_Array_Received[2].0;
			
			//Go to Next Step
			timer_Timeout.IN := FALSE;
			fbMBRead_FC3.bExecute := FALSE;
			timer_Delay.IN := FALSE;		
			iStateModbusRead := 30;
		END_IF	

		//Error or Timeout
		IF FPError_FC_3.Q THEN 
			iStateModbusError := 300;
			int_FC3Error := int_FC3Error+1;
		ELSIF timer_Timeout.Q THEN  
			timer_Timeout.IN := FALSE; 	
			iStateModbusError := 300;
			int_TimeoutError := int_TimeoutError+1;
		END_IF
		
	
	30://Wait and go to step 1
		//1 because 0 is the Init Step for Read
		timer_Wait.IN := TRUE;
		
		IF timer_Wait.Q = TRUE THEN
			iStateModbusRead := 0;
			timer_Wait.IN :=FALSE;
		END_IF

			
		
		//Error on Master, changes on Inputs or Timeout
		IF timer_Timeout.Q THEN 
			iStateModbusError := 300; 
		END_IF
	
END_CASE

(* wait timer*)

timer_Wait(PT:=T#1S);


(*------------------------------------------------------------------Error and Warning----------------------------------------------------------------------------*)	
 
timer_Connection_ok			(In:=int_Data_Received<>int_Data_Received_old,PT:=T#10S);
timer_Connection_ok_TOF		(In:=NOT(int_Data_Received<>int_Data_Received_old) AND int_Data_Received>3 ,PT:=T#20S);
int_Data_Received_old:=int_Data_Received;
m_PollSuccessful:=NOT timer_Connection_ok.Q AND timer_Connection_ok_TOF.Q ;

(*------------------------------------------------------------------------------------------Modbus TCP Functions---------------------------------------------------------------------------------------------*)

fbMBRead_FC3(	sIPAddr:= str_IPAdress, 
				nTCPPort:= uint_port,
				cbLength:= SIZEOF(arrBuffer_FC3), 
				pDestAddr:= ADR(arrBuffer_FC3), 
				tTimeout:= T#10S,
				nErrId => udint_Error_ID);

FPError_FC_3(CLK:= fbMBRead_FC3.bError, Q=> );		

(*------------------------------------------------------------------------------------------State Machine Error---------------------------------------------------------------------------------------------*)	

CASE iStateModbusError OF
	
	300://Error
		timer_Wait.IN :=TRUE;
		timer_Delay.IN := FALSE;
		fbMBRead_FC3.bExecute := FALSE;
		m_MBTCPError := TRUE; 		
		m_Poll_ok:=FALSE;
		int_Data_Received:=0;
				//Restart from new with the Read out part after an Error
		IF timer_Wait.Q = TRUE THEN
			iStateModbusRead := 0;	
			iStateModbusError := 0;
			timer_Wait.IN :=FALSE;
			timer_Timeout.IN := FALSE;
		END_IF		
							
END_CASE

END_FUNCTION_BLOCK

// ---- POUs/prgE5.TcPOU
PROGRAM prgE5
VAR
	FB_Read_MB :FB_ModBus_100Registers_FC3;
	m_Enable: BOOL ;
	str_IP: STRING(15):= '192.168.8.4';
	word_Adress: WORD;
	usint_Quantity: USINT;
	byte_slaveID: BYTE;

	lr_RC_Anlage_Freq 			: LREAL;		//{#lynus.ag#()}
	lr_RC_Anlage_L1N 			: LREAL;		//{#lynus.ag#()}
	lr_RC_Anlage_L2N 			: LREAL;		//{#lynus.ag#()}
	lr_RC_Anlage_L3N 			: LREAL;		//{#lynus.ag#()}
	lr_RC_Anlage_L1L2 			: LREAL;		//{#lynus.ag#()}
	lr_RC_Anlage_L2L3 			: LREAL;		//{#lynus.ag#()}
	lr_RC_Anlage_L3L1 			: LREAL;		//{#lynus.ag#()}
	lr_RC_Anlage_I1 			: LREAL;		//{#lynus.ag#()}
	lr_RC_Anlage_I2 			: LREAL;		//{#lynus.ag#()}
	lr_RC_Anlage_I3 			: LREAL;		//{#lynus.ag#()}
	lr_RC_Anlage_N 				: LREAL;		//{#lynus.ag#()}
	lr_RC_Anlage_S 				: LREAL;		//{#lynus.ag#()}
	lr_RC_Anlage_P 				: LREAL;		//{#lynus.ag#()}
	lr_RC_Anlage_Q 				: LREAL;		//{#lynus.ag#()}
	lr_RC_Anlage_PF 			: LREAL;		//{#lynus.ag#()}
	
	lr_RC_Trommel_Freq 			: LREAL;		//{#lynus.ag#()}
	lr_RC_Trommel_L1N 			: LREAL;		//{#lynus.ag#()}
	lr_RC_Trommel_L2N 			: LREAL;		//{#lynus.ag#()}
	lr_RC_Trommel_L3N 			: LREAL;		//{#lynus.ag#()}
	lr_RC_Trommel_L1L2 			: LREAL;		//{#lynus.ag#()}
	lr_RC_Trommel_L2L3 			: LREAL;		//{#lynus.ag#()}
	lr_RC_Trommel_L3L1 			: LREAL;		//{#lynus.ag#()}
	lr_RC_Trommel_I1 			: LREAL;		//{#lynus.ag#()}
	lr_RC_Trommel_I2 			: LREAL;		//{#lynus.ag#()}
	lr_RC_Trommel_I3 			: LREAL;		//{#lynus.ag#()}
	lr_RC_Trommel_N 			: LREAL;		//{#lynus.ag#()}
	lr_RC_Trommel_S 			: LREAL;		//{#lynus.ag#()}
	lr_RC_Trommel_P 			: LREAL;		//{#lynus.ag#()}
	lr_RC_Trommel_Q 			: LREAL;		//{#lynus.ag#()}
	lr_RC_Trommel_PF 			: LREAL;		//{#lynus.ag#()}
	
	lr_GasmessungRTMenge_m3h 	: LREAL;		//{#lynus.ag#()}
	lr_GasmessungRTTemp_C 		: LREAL;		//{#lynus.ag#()}
	lr_GasmessungRTDruck_bar 	: LREAL;		//{#lynus.ag#()}
	
	m_Brennerstart_RC	 		: BOOL;			//{#lynus.ag#()}
	m_Oelzaehler	 			: BOOL;			//{#lynus.ag#()}
	
	FB_Read_Socomec_I61 	: FB_Socomec_I61;
	FB_Read_Socomec_IO20	: FB_Socomec_IO20;
	FB_Read_Socomec_IO10	: FB_Socomec_IO10;
	i_State_ModbusCall: INT;				
	ton_TimeOutState: ton;
	tof_TimeOut_Active: tof;
	i_State_ModbusCall_old: INT;
	int_errorCount: INT;
	m_TimeOutActive: BOOL;					//{#lynus.ag#()}
	i_State_ErrorActive: INT;				//{#lynus.ag#()}
END_VAR

CASE i_State_ModbusCall OF
	0: 	// wait state
		i_State_ModbusCall := 10;
	
	10:	// first Modbus Poll Call
		FB_Read_Socomec_I61.m_Start := TRUE;
		FB_Read_Socomec_I61.byte_slaveID := 43;
		FB_Read_Socomec_I61.w_Adress := 18442;
		i_State_ModbusCall := i_State_ModbusCall + 1;
	
	11: // wait for received data
		FB_Read_Socomec_I61.m_Start := FALSE;
		IF FB_Read_Socomec_I61.iStateModbusRead = 30 THEN
			lr_RC_Anlage_Freq	:=		FB_Read_Socomec_I61.lr_Freq_Hz	;	
			lr_RC_Anlage_L1N	:=		FB_Read_Socomec_I61.lr_L1N_V	;	
			lr_RC_Anlage_L2N	:=		FB_Read_Socomec_I61.lr_L2N_V	;	
			lr_RC_Anlage_L3N	:=		FB_Read_Socomec_I61.lr_L3N_V	;	
			lr_RC_Anlage_L1L2	:=		FB_Read_Socomec_I61.lr_L1L2_V	;	
			lr_RC_Anlage_L2L3	:=		FB_Read_Socomec_I61.lr_L2L3_V	;	
			lr_RC_Anlage_L3L1	:=		FB_Read_Socomec_I61.lr_L3L1_V	;	
			lr_RC_Anlage_I1		:=		FB_Read_Socomec_I61.lr_I1_A		;	
			lr_RC_Anlage_I2		:=		FB_Read_Socomec_I61.lr_I2_A		;	
			lr_RC_Anlage_I3		:=		FB_Read_Socomec_I61.lr_I3_A		;	
			lr_RC_Anlage_N		:=		FB_Read_Socomec_I61.lr_N_A		;	
			lr_RC_Anlage_P		:=		FB_Read_Socomec_I61.lr_P_kW		;	
			lr_RC_Anlage_Q		:=		FB_Read_Socomec_I61.lr_Q_kVAr	;	
			lr_RC_Anlage_S		:=		FB_Read_Socomec_I61.lr_S_kVA	;	
			lr_RC_Anlage_PF		:=		FB_Read_Socomec_I61.lr_PF		;		
			
			i_State_ModbusCall := i_State_ModbusCall +1;
		END_IF            
		IF FB_Read_Socomec_I61.iStateModbusError = 300 OR ton_TimeOutState.Q THEN
			i_State_ModbusCall := i_State_ModbusCall +1;
		END_IF
	
	12: // wait for FB_Read_Socomec_I61 to be in state 0
		IF FB_Read_Socomec_I61.iStateModbusRead = 0 OR ton_TimeOutState.Q THEN
			i_State_ModbusCall := i_State_ModbusCall + 8;
		END_IF
	
	20:	// next Modbus Poll Call
		FB_Read_Socomec_I61.m_Start := TRUE;
		FB_Read_Socomec_I61.byte_slaveID := 43;
		FB_Read_Socomec_I61.w_Adress := 20490;
		i_State_ModbusCall := i_State_ModbusCall + 1;
	
	21: // wait for received data
		FB_Read_Socomec_I61.m_Start := FALSE;
		IF FB_Read_Socomec_I61.iStateModbusRead = 30 THEN
			lr_RC_Trommel_Freq		:=		FB_Read_Socomec_I61.lr_Freq_Hz	;	
			lr_RC_Trommel_L1N		:=		FB_Read_Socomec_I61.lr_L1N_V	;	
			lr_RC_Trommel_L2N		:=		FB_Read_Socomec_I61.lr_L2N_V	;	
			lr_RC_Trommel_L3N		:=		FB_Read_Socomec_I61.lr_L3N_V	;	
			lr_RC_Trommel_L1L2		:=		FB_Read_Socomec_I61.lr_L1L2_V	;	
			lr_RC_Trommel_L2L3		:=		FB_Read_Socomec_I61.lr_L2L3_V	;	
			lr_RC_Trommel_L3L1		:=		FB_Read_Socomec_I61.lr_L3L1_V	;	
			lr_RC_Trommel_I1		:=		FB_Read_Socomec_I61.lr_I1_A		;	
			lr_RC_Trommel_I2		:=		FB_Read_Socomec_I61.lr_I2_A		;	
			lr_RC_Trommel_I3		:=		FB_Read_Socomec_I61.lr_I3_A		;	
			lr_RC_Trommel_N			:=		FB_Read_Socomec_I61.lr_N_A		;	
			lr_RC_Trommel_P			:=		FB_Read_Socomec_I61.lr_P_kW		;	
			lr_RC_Trommel_Q			:=		FB_Read_Socomec_I61.lr_Q_kVAr	;	
			lr_RC_Trommel_S			:=		FB_Read_Socomec_I61.lr_S_kVA	;	
			lr_RC_Trommel_PF		:=		FB_Read_Socomec_I61.lr_PF		;		
			
			i_State_ModbusCall := i_State_ModbusCall +1;
		END_IF            
		IF FB_Read_Socomec_I61.iStateModbusError = 300 OR ton_TimeOutState.Q THEN
			i_State_ModbusCall := i_State_ModbusCall +1;
		END_IF
	
	22: // wait for FB_Read_Socomec_I61 to be in state 0
		IF FB_Read_Socomec_I61.iStateModbusRead = 0 OR ton_TimeOutState.Q THEN
			i_State_ModbusCall := i_State_ModbusCall + 8;
		END_IF
	
	30:	// next Modbus Poll Call		first IO20 call
		FB_Read_Socomec_IO20.m_Start := TRUE;
		FB_Read_Socomec_IO20.byte_slaveID := 44;
		FB_Read_Socomec_IO20.w_Adress := 11589;
		i_State_ModbusCall := i_State_ModbusCall + 1;
	
	31: // wait for received data
		FB_Read_Socomec_IO20.m_Start := FALSE;
		IF FB_Read_Socomec_IO20.iStateModbusRead = 30 THEN
			lr_GasmessungRTMenge_m3h := LIMIT(0,2150.0/16.0*(FB_Read_Socomec_IO20.lr_Value_mA-4),2150);		// 4-20mA = 0-2150 m3/h
			i_State_ModbusCall := i_State_ModbusCall +1;
		END_IF            
		IF FB_Read_Socomec_I61.iStateModbusError = 300 OR ton_TimeOutState.Q THEN
			i_State_ModbusCall := i_State_ModbusCall +1;
		END_IF
	
	32: // wait for FB_Read_Socomec_IO20 to be in state 0
		IF FB_Read_Socomec_IO20.iStateModbusRead = 0 OR ton_TimeOutState.Q THEN
			i_State_ModbusCall := i_State_ModbusCall + 8;
		END_IF
		
	40:	// next Modbus Poll Call		second IO20 call
		FB_Read_Socomec_IO20.m_Start := TRUE;
		FB_Read_Socomec_IO20.byte_slaveID := 44;
		FB_Read_Socomec_IO20.w_Adress := 11621;
		i_State_ModbusCall := i_State_ModbusCall + 1;
	
	41: // wait for received data
		FB_Read_Socomec_IO20.m_Start := FALSE;
		IF FB_Read_Socomec_IO20.iStateModbusRead = 30 THEN
			lr_GasmessungRTTemp_C := LIMIT(-20,100.0/16.0*(FB_Read_Socomec_IO20.lr_Value_mA-4)-20,80);		// 4-20mA = -20-80 °C
				
			i_State_ModbusCall := i_State_ModbusCall +1;
		END_IF            
		IF FB_Read_Socomec_IO20.iStateModbusError = 300 OR ton_TimeOutState.Q THEN
			i_State_ModbusCall := i_State_ModbusCall +1;
		END_IF
	
	42: // wait for FB_Read_Socomec_IO20 to be in state 0
		IF FB_Read_Socomec_IO20.iStateModbusRead = 0 OR ton_TimeOutState.Q THEN
			i_State_ModbusCall := i_State_ModbusCall + 8;
		END_IF
	50:	// next Modbus Poll Call		third IO20 call
		FB_Read_Socomec_IO20.m_Start := TRUE;
		FB_Read_Socomec_IO20.byte_slaveID := 45;
		FB_Read_Socomec_IO20.w_Adress := 11589;
		i_State_ModbusCall := i_State_ModbusCall + 1;
	
	51: // wait for received data
		FB_Read_Socomec_IO20.m_Start := FALSE;
		IF FB_Read_Socomec_IO20.iStateModbusRead = 30 THEN
			lr_GasmessungRTDruck_bar :=	LIMIT(0,(5.0/16.0) * (FB_Read_Socomec_IO20.lr_Value_mA-4),5);		// 4-20mA = 0-5 bar
			i_State_ModbusCall := i_State_ModbusCall +1;
		END_IF            
		IF FB_Read_Socomec_IO20.iStateModbusError = 300 OR ton_TimeOutState.Q THEN
			i_State_ModbusCall := i_State_ModbusCall +1;
		END_IF
	
	52: // wait for FB_Read_Socomec_IO20 to be in state 0
		IF FB_Read_Socomec_IO20.iStateModbusRead = 0 OR ton_TimeOutState.Q THEN
			i_State_ModbusCall := i_State_ModbusCall + 8;
		END_IF	

	60:	// next Modbus Poll Call		first IO10 call
		FB_Read_Socomec_IO10.m_Start := TRUE;
		FB_Read_Socomec_IO10.byte_slaveID := 46;
		FB_Read_Socomec_IO10.w_Adress := 11520;
		i_State_ModbusCall := i_State_ModbusCall + 1;
	
	61: // wait for received data
		FB_Read_Socomec_IO10.m_Start := FALSE;
		IF FB_Read_Socomec_IO10.iStateModbusRead = 30 THEN
			m_Brennerstart_RC := FB_Read_Socomec_IO10.m_Input_Active;		
				
			i_State_ModbusCall := i_State_ModbusCall +1;
		END_IF            
		IF FB_Read_Socomec_IO10.iStateModbusError = 300 OR ton_TimeOutState.Q THEN
			i_State_ModbusCall := i_State_ModbusCall +1;
		END_IF
	
	62: // wait for FB_Read_Socomec_IO10 to be in state 0
		IF FB_Read_Socomec_IO10.iStateModbusRead = 0 OR ton_TimeOutState.Q THEN
			i_State_ModbusCall := i_State_ModbusCall + 8;
		END_IF

	70:	// next Modbus Poll Call		first IO10 call
		FB_Read_Socomec_IO10.m_Start := TRUE;
		FB_Read_Socomec_IO10.byte_slaveID := 46;
		FB_Read_Socomec_IO10.w_Adress := 11524;
		i_State_ModbusCall := i_State_ModbusCall + 1;
	
	71: // wait for received data
		FB_Read_Socomec_IO10.m_Start := FALSE;
		IF FB_Read_Socomec_IO10.iStateModbusRead = 30 THEN
			m_Oelzaehler := FB_Read_Socomec_IO10.m_Input_Active;		
				
			i_State_ModbusCall := i_State_ModbusCall +1;
		END_IF            
		IF FB_Read_Socomec_IO10.iStateModbusError = 300 OR ton_TimeOutState.Q THEN
			i_State_ModbusCall := i_State_ModbusCall +1;
		END_IF
	
	72: // wait for FB_Read_Socomec_IO10 to be in state 0
		IF FB_Read_Socomec_IO10.iStateModbusRead = 0 OR ton_TimeOutState.Q THEN
			i_State_ModbusCall := i_State_ModbusCall + 8;
		END_IF		
		
	80: 
		i_State_ModbusCall := 0;
END_CASE

ton_TimeOutState(	IN:= i_State_ModbusCall = i_State_ModbusCall_old, 
					PT:= T#30S, 
					Q=> , 
					ET=> );

i_State_ModbusCall_old := i_State_ModbusCall; 

IF ton_TimeOutState.Q THEN
//	i_State_ModbusCall := 0;
	int_errorCount := int_errorCount  + 1; 
END_IF


tof_TimeOut_Active(	IN:= ton_TimeOutState.Q, 
					PT:=	T#5S , 
					Q=> m_TimeOutActive, 
					ET=> );
IF tof_TimeOut_Active.Q THEN
	 i_State_ErrorActive := i_State_ModbusCall; 
END_IF


FB_Read_Socomec_I61(
	m_Start:= , 
	str_IPAdress:= str_IP , 
	w_Adress:= , 
	uint_port:= , 
	byte_slaveID:= , 
	m_PollSuccessful=> , 
	lr_Freq_Hz=> , 
	lr_L1N_V=> , 
	lr_L2N_V=> , 
	lr_L3N_V=> , 
	lr_L1L2_V=> , 
	lr_L2L3_V=> , 
	lr_L3L1_V=> , 
	lr_I1_A=> , 
	lr_I2_A=> , 
	lr_I3_A=> , 
	lr_N_A=> , 
	lr_P_kW=> , 
	lr_Q_kVAr=> , 
	lr_S_kVA=> , 
	lr_PF=> , 
	udint_Error_ID=> );

FB_Read_Socomec_IO20(
	m_Start:= , 
	str_IPAdress:= str_IP, 
	w_Adress:= , 
	uint_port:= , 
	byte_slaveID:= , 
	m_PollSuccessful=> , 
	lr_Value_mA=> , 
	udint_Error_ID=> );	
	
FB_Read_Socomec_IO10(
	m_Start:= , 
	str_IPAdress:= str_IP , 
	w_Adress:= , 
	uint_port:= , 
	byte_slaveID:= , 
	m_PollSuccessful=> , 
	m_Input_Active=> , 
	udint_Error_ID=> );	

FB_Read_MB(
	m_Enable:= m_Enable, 
	str_IPAdress:= str_IP,
	w_Adress:= word_Adress, 
	usint_Quantity:= usint_Quantity, 
	byte_slaveID:=byte_slaveID,
	uint_port := ,
	m_PollSuccessful=> , 
	w_Array_Received=> , 
	udint_Error_ID=> );

END_PROGRAM

// ---- POUs/prgE9.TcPOU
PROGRAM prgE9
VAR
	FB_Read_MB :FB_ModBus_100Registers_FC3;
	m_Enable: BOOL;
	str_IP: STRING(15):= '192.168.8.3';
	word_Adress: WORD;
	usint_Quantity: USINT;
	byte_slaveID: BYTE;
	
	lr_Bitumentank_1_Freq 			: LREAL;		//{#lynus.ag#()}
	lr_Bitumentank_1_L1N 			: LREAL;		//{#lynus.ag#()}
	lr_Bitumentank_1_L2N 			: LREAL;		//{#lynus.ag#()}
	lr_Bitumentank_1_L3N 			: LREAL;		//{#lynus.ag#()}
	lr_Bitumentank_1_L1L2 			: LREAL;		//{#lynus.ag#()}
	lr_Bitumentank_1_L2L3 			: LREAL;		//{#lynus.ag#()}
	lr_Bitumentank_1_L3L1 			: LREAL;		//{#lynus.ag#()}
	lr_Bitumentank_1_I1 			: LREAL;		//{#lynus.ag#()}
	lr_Bitumentank_1_I2 			: LREAL;		//{#lynus.ag#()}
	lr_Bitumentank_1_I3 			: LREAL;		//{#lynus.ag#()}
	lr_Bitumentank_1_N 				: LREAL;		//{#lynus.ag#()}
	lr_Bitumentank_1_S 				: LREAL;		//{#lynus.ag#()}
	lr_Bitumentank_1_P 				: LREAL;		//{#lynus.ag#()}
	lr_Bitumentank_1_Q 				: LREAL;		//{#lynus.ag#()}
	lr_Bitumentank_1_PF 			: LREAL;		//{#lynus.ag#()}
	
	lr_Bitumentank_2_Freq 			: LREAL;		//{#lynus.ag#()}
	lr_Bitumentank_2_L1N 			: LREAL;		//{#lynus.ag#()}
	lr_Bitumentank_2_L2N 			: LREAL;		//{#lynus.ag#()}
	lr_Bitumentank_2_L3N 			: LREAL;		//{#lynus.ag#()}
	lr_Bitumentank_2_L1L2 			: LREAL;		//{#lynus.ag#()}
	lr_Bitumentank_2_L2L3 			: LREAL;		//{#lynus.ag#()}
	lr_Bitumentank_2_L3L1 			: LREAL;		//{#lynus.ag#()}
	lr_Bitumentank_2_I1 			: LREAL;		//{#lynus.ag#()}
	lr_Bitumentank_2_I2 			: LREAL;		//{#lynus.ag#()}
	lr_Bitumentank_2_I3 			: LREAL;		//{#lynus.ag#()}
	lr_Bitumentank_2_N 				: LREAL;		//{#lynus.ag#()}
	lr_Bitumentank_2_S 				: LREAL;		//{#lynus.ag#()}
	lr_Bitumentank_2_P 				: LREAL;		//{#lynus.ag#()}
	lr_Bitumentank_2_Q 				: LREAL;		//{#lynus.ag#()}
	lr_Bitumentank_2_PF 			: LREAL;		//{#lynus.ag#()}
	
	lr_Bitumentank_3_Freq 			: LREAL;		//{#lynus.ag#()}
	lr_Bitumentank_3_L1N 			: LREAL;		//{#lynus.ag#()}
	lr_Bitumentank_3_L2N 			: LREAL;		//{#lynus.ag#()}
	lr_Bitumentank_3_L3N 			: LREAL;		//{#lynus.ag#()}
	lr_Bitumentank_3_L1L2 			: LREAL;		//{#lynus.ag#()}
	lr_Bitumentank_3_L2L3 			: LREAL;		//{#lynus.ag#()}
	lr_Bitumentank_3_L3L1 			: LREAL;		//{#lynus.ag#()}
	lr_Bitumentank_3_I1 			: LREAL;		//{#lynus.ag#()}
	lr_Bitumentank_3_I2 			: LREAL;		//{#lynus.ag#()}
	lr_Bitumentank_3_I3 			: LREAL;		//{#lynus.ag#()}
	lr_Bitumentank_3_N 				: LREAL;		//{#lynus.ag#()}
	lr_Bitumentank_3_S 				: LREAL;		//{#lynus.ag#()}
	lr_Bitumentank_3_P 				: LREAL;		//{#lynus.ag#()}
	lr_Bitumentank_3_Q 				: LREAL;		//{#lynus.ag#()}
	lr_Bitumentank_3_PF 			: LREAL;		//{#lynus.ag#()}
	
	lr_Bitumentank_4_Freq 			: LREAL;		//{#lynus.ag#()}
	lr_Bitumentank_4_L1N 			: LREAL;		//{#lynus.ag#()}
	lr_Bitumentank_4_L2N 			: LREAL;		//{#lynus.ag#()}
	lr_Bitumentank_4_L3N 			: LREAL;		//{#lynus.ag#()}
	lr_Bitumentank_4_L1L2 			: LREAL;		//{#lynus.ag#()}
	lr_Bitumentank_4_L2L3 			: LREAL;		//{#lynus.ag#()}
	lr_Bitumentank_4_L3L1 			: LREAL;		//{#lynus.ag#()}
	lr_Bitumentank_4_I1 			: LREAL;		//{#lynus.ag#()}
	lr_Bitumentank_4_I2 			: LREAL;		//{#lynus.ag#()}
	lr_Bitumentank_4_I3 			: LREAL;		//{#lynus.ag#()}
	lr_Bitumentank_4_N 				: LREAL;		//{#lynus.ag#()}
	lr_Bitumentank_4_S 				: LREAL;		//{#lynus.ag#()}
	lr_Bitumentank_4_P 				: LREAL;		//{#lynus.ag#()}
	lr_Bitumentank_4_Q 				: LREAL;		//{#lynus.ag#()}
	lr_Bitumentank_4_PF 			: LREAL;		//{#lynus.ag#()}
	
	lr_Bitumenfuellpumpe_1_Freq 	: LREAL;		//{#lynus.ag#()}
	lr_Bitumenfuellpumpe_1_L1N 		: LREAL;		//{#lynus.ag#()}
	lr_Bitumenfuellpumpe_1_L2N 		: LREAL;		//{#lynus.ag#()}
	lr_Bitumenfuellpumpe_1_L3N 		: LREAL;		//{#lynus.ag#()}
	lr_Bitumenfuellpumpe_1_L1L2 	: LREAL;		//{#lynus.ag#()}
	lr_Bitumenfuellpumpe_1_L2L3 	: LREAL;		//{#lynus.ag#()}
	lr_Bitumenfuellpumpe_1_L3L1		: LREAL;		//{#lynus.ag#()}
	lr_Bitumenfuellpumpe_1_I1 		: LREAL;		//{#lynus.ag#()}
	lr_Bitumenfuellpumpe_1_I2 		: LREAL;		//{#lynus.ag#()}
	lr_Bitumenfuellpumpe_1_I3 		: LREAL;		//{#lynus.ag#()}
	lr_Bitumenfuellpumpe_1_N 		: LREAL;		//{#lynus.ag#()}
	lr_Bitumenfuellpumpe_1_S 		: LREAL;		//{#lynus.ag#()}
	lr_Bitumenfuellpumpe_1_P 		: LREAL;		//{#lynus.ag#()}
	lr_Bitumenfuellpumpe_1_Q 		: LREAL;		//{#lynus.ag#()}
	lr_Bitumenfuellpumpe_1_PF 		: LREAL;		//{#lynus.ag#()}

	lr_Dosierpumpe_1_Freq 			: LREAL;		//{#lynus.ag#()}
	lr_Dosierpumpe_1_L1N 			: LREAL;		//{#lynus.ag#()}
	lr_Dosierpumpe_1_L2N 			: LREAL;		//{#lynus.ag#()}
	lr_Dosierpumpe_1_L3N 			: LREAL;		//{#lynus.ag#()}
	lr_Dosierpumpe_1_L1L2 			: LREAL;		//{#lynus.ag#()}
	lr_Dosierpumpe_1_L2L3 			: LREAL;		//{#lynus.ag#()}
	lr_Dosierpumpe_1_L3L1 			: LREAL;		//{#lynus.ag#()}
	lr_Dosierpumpe_1_I1 			: LREAL;		//{#lynus.ag#()}
	lr_Dosierpumpe_1_I2 			: LREAL;		//{#lynus.ag#()}
	lr_Dosierpumpe_1_I3 			: LREAL;		//{#lynus.ag#()}
	lr_Dosierpumpe_1_N 				: LREAL;		//{#lynus.ag#()}
	lr_Dosierpumpe_1_S 				: LREAL;		//{#lynus.ag#()}
	lr_Dosierpumpe_1_P 				: LREAL;		//{#lynus.ag#()}
	lr_Dosierpumpe_1_Q 				: LREAL;		//{#lynus.ag#()}
	lr_Dosierpumpe_1_PF 			: LREAL;		//{#lynus.ag#()}

	lr_Dosierpumpe_2_Freq 			: LREAL;		//{#lynus.ag#()}
	lr_Dosierpumpe_2_L1N 			: LREAL;		//{#lynus.ag#()}
	lr_Dosierpumpe_2_L2N 			: LREAL;		//{#lynus.ag#()}
	lr_Dosierpumpe_2_L3N 			: LREAL;		//{#lynus.ag#()}
	lr_Dosierpumpe_2_L1L2 			: LREAL;		//{#lynus.ag#()}
	lr_Dosierpumpe_2_L2L3 			: LREAL;		//{#lynus.ag#()}
	lr_Dosierpumpe_2_L3L1 			: LREAL;		//{#lynus.ag#()}
	lr_Dosierpumpe_2_I1 			: LREAL;		//{#lynus.ag#()}
	lr_Dosierpumpe_2_I2 			: LREAL;		//{#lynus.ag#()}
	lr_Dosierpumpe_2_I3 			: LREAL;		//{#lynus.ag#()}
	lr_Dosierpumpe_2_N 				: LREAL;		//{#lynus.ag#()}
	lr_Dosierpumpe_2_S 				: LREAL;		//{#lynus.ag#()}
	lr_Dosierpumpe_2_P 				: LREAL;		//{#lynus.ag#()}
	lr_Dosierpumpe_2_Q 				: LREAL;		//{#lynus.ag#()}
	lr_Dosierpumpe_2_PF 			: LREAL;		//{#lynus.ag#()}
	
	m_Bitumenfuellpumpe_1	 		: BOOL;			//{#lynus.ag#()}
	
	FB_Read_Socomec_I61 	: FB_Socomec_I61;
	FB_Read_Socomec_I31 	: FB_Socomec_I31;
	FB_Read_Socomec_IO10	: FB_Socomec_IO10;
	i_State_ModbusCall: INT;				
	ton_TimeOutState: ton;
	tof_TimeOut_Active: tof;
	i_State_ModbusCall_old: INT;
	int_errorCount: INT;
	m_TimeOutActive: BOOL;					//{#lynus.ag#()}
	i_State_ErrorActive: INT;				//{#lynus.ag#()}
END_VAR

CASE i_State_ModbusCall OF
	0: 	// wait state
		i_State_ModbusCall := 10;
	
	10:	// first Modbus Poll Call
		FB_Read_Socomec_I61.m_Start := TRUE;
		FB_Read_Socomec_I61.byte_slaveID := 26;
		FB_Read_Socomec_I61.w_Adress := 18442;
		i_State_ModbusCall := i_State_ModbusCall + 1;
	
	11: // wait for received data
		FB_Read_Socomec_I61.m_Start := FALSE;
		IF FB_Read_Socomec_I61.iStateModbusRead = 30 THEN
			lr_Bitumentank_4_Freq	:=		FB_Read_Socomec_I61.lr_Freq_Hz	;	
			lr_Bitumentank_4_L1N	:=		FB_Read_Socomec_I61.lr_L1N_V	;	
			lr_Bitumentank_4_L2N	:=		FB_Read_Socomec_I61.lr_L2N_V	;	
			lr_Bitumentank_4_L3N	:=		FB_Read_Socomec_I61.lr_L3N_V	;	
			lr_Bitumentank_4_L1L2	:=		FB_Read_Socomec_I61.lr_L1L2_V	;	
			lr_Bitumentank_4_L2L3	:=		FB_Read_Socomec_I61.lr_L2L3_V	;	
			lr_Bitumentank_4_L3L1	:=		FB_Read_Socomec_I61.lr_L3L1_V	;	
			lr_Bitumentank_4_I1		:=		FB_Read_Socomec_I61.lr_I1_A		;	
			lr_Bitumentank_4_I2		:=		FB_Read_Socomec_I61.lr_I2_A		;	
			lr_Bitumentank_4_I3		:=		FB_Read_Socomec_I61.lr_I3_A		;	
			lr_Bitumentank_4_N		:=		FB_Read_Socomec_I61.lr_N_A		;	
			lr_Bitumentank_4_P		:=		FB_Read_Socomec_I61.lr_P_kW		;	
			lr_Bitumentank_4_Q		:=		FB_Read_Socomec_I61.lr_Q_kVAr	;	
			lr_Bitumentank_4_S		:=		FB_Read_Socomec_I61.lr_S_kVA	;	
			lr_Bitumentank_4_PF		:=		FB_Read_Socomec_I61.lr_PF		;		
			
			i_State_ModbusCall := i_State_ModbusCall +1;
		END_IF            
		IF FB_Read_Socomec_I61.iStateModbusError = 300 OR ton_TimeOutState.Q THEN
			i_State_ModbusCall := i_State_ModbusCall +1;
		END_IF
	
	12: // wait for FB_Read_Socomec_I61 to be in state 0
		IF FB_Read_Socomec_I61.iStateModbusRead = 0 OR ton_TimeOutState.Q THEN
			i_State_ModbusCall := i_State_ModbusCall + 8;
		END_IF

	20:	// next Modbus Poll Call
		FB_Read_Socomec_I61.m_Start := TRUE;
		FB_Read_Socomec_I61.byte_slaveID := 27;
		FB_Read_Socomec_I61.w_Adress := 18442;
		i_State_ModbusCall := i_State_ModbusCall + 1;
	
	21: // wait for received data
		FB_Read_Socomec_I61.m_Start := FALSE;
		IF FB_Read_Socomec_I61.iStateModbusRead = 30 THEN
			lr_Dosierpumpe_1_Freq		:=		FB_Read_Socomec_I61.lr_Freq_Hz	;	
			lr_Dosierpumpe_1_L1N		:=		FB_Read_Socomec_I61.lr_L1N_V	;	
			lr_Dosierpumpe_1_L2N		:=		FB_Read_Socomec_I61.lr_L2N_V	;	
			lr_Dosierpumpe_1_L3N		:=		FB_Read_Socomec_I61.lr_L3N_V	;	
			lr_Dosierpumpe_1_L1L2		:=		FB_Read_Socomec_I61.lr_L1L2_V	;	
			lr_Dosierpumpe_1_L2L3		:=		FB_Read_Socomec_I61.lr_L2L3_V	;	
			lr_Dosierpumpe_1_L3L1		:=		FB_Read_Socomec_I61.lr_L3L1_V	;	
			lr_Dosierpumpe_1_I1			:=		FB_Read_Socomec_I61.lr_I1_A		;	
			lr_Dosierpumpe_1_I2			:=		FB_Read_Socomec_I61.lr_I2_A		;	
			lr_Dosierpumpe_1_I3			:=		FB_Read_Socomec_I61.lr_I3_A		;	
			lr_Dosierpumpe_1_N			:=		FB_Read_Socomec_I61.lr_N_A		;	
			lr_Dosierpumpe_1_P			:=		FB_Read_Socomec_I61.lr_P_kW		;	
			lr_Dosierpumpe_1_Q			:=		FB_Read_Socomec_I61.lr_Q_kVAr	;	
			lr_Dosierpumpe_1_S			:=		FB_Read_Socomec_I61.lr_S_kVA	;	
			lr_Dosierpumpe_1_PF			:=		FB_Read_Socomec_I61.lr_PF		;		
			
			i_State_ModbusCall := i_State_ModbusCall +1;
		END_IF            
		IF FB_Read_Socomec_I61.iStateModbusError = 300 OR ton_TimeOutState.Q THEN
			i_State_ModbusCall := i_State_ModbusCall +1;
		END_IF
	
	22: // wait for FB_Read_Socomec_I61 to be in state 0
		IF FB_Read_Socomec_I61.iStateModbusRead = 0 OR ton_TimeOutState.Q THEN
			i_State_ModbusCall := i_State_ModbusCall + 8;
		END_IF
	
	30:	// next Modbus Poll Call
		FB_Read_Socomec_I61.m_Start := TRUE;
		FB_Read_Socomec_I61.byte_slaveID := 26;
		FB_Read_Socomec_I61.w_Adress := 20490;
		i_State_ModbusCall := i_State_ModbusCall + 1;
	
	31: // wait for received data
		FB_Read_Socomec_I61.m_Start := FALSE;
		IF FB_Read_Socomec_I61.iStateModbusRead = 30 THEN
			lr_Bitumenfuellpumpe_1_Freq		:=		FB_Read_Socomec_I61.lr_Freq_Hz	;	
			lr_Bitumenfuellpumpe_1_L1N		:=		FB_Read_Socomec_I61.lr_L1N_V	;	
			lr_Bitumenfuellpumpe_1_L2N		:=		FB_Read_Socomec_I61.lr_L2N_V	;	
			lr_Bitumenfuellpumpe_1_L3N		:=		FB_Read_Socomec_I61.lr_L3N_V	;	
			lr_Bitumenfuellpumpe_1_L1L2		:=		FB_Read_Socomec_I61.lr_L1L2_V	;	
			lr_Bitumenfuellpumpe_1_L2L3		:=		FB_Read_Socomec_I61.lr_L2L3_V	;	
			lr_Bitumenfuellpumpe_1_L3L1		:=		FB_Read_Socomec_I61.lr_L3L1_V	;	
			lr_Bitumenfuellpumpe_1_I1		:=		FB_Read_Socomec_I61.lr_I1_A		;	
			lr_Bitumenfuellpumpe_1_I2		:=		FB_Read_Socomec_I61.lr_I2_A		;	
			lr_Bitumenfuellpumpe_1_I3		:=		FB_Read_Socomec_I61.lr_I3_A		;	
			lr_Bitumenfuellpumpe_1_N		:=		FB_Read_Socomec_I61.lr_N_A		;	
			lr_Bitumenfuellpumpe_1_P		:=		FB_Read_Socomec_I61.lr_P_kW		;	
			lr_Bitumenfuellpumpe_1_Q		:=		FB_Read_Socomec_I61.lr_Q_kVAr	;	
			lr_Bitumenfuellpumpe_1_S		:=		FB_Read_Socomec_I61.lr_S_kVA	;	
			lr_Bitumenfuellpumpe_1_PF		:=		FB_Read_Socomec_I61.lr_PF		;		
			
			i_State_ModbusCall := i_State_ModbusCall +1;
		END_IF            
		IF FB_Read_Socomec_I61.iStateModbusError = 300 OR ton_TimeOutState.Q THEN
			i_State_ModbusCall := i_State_ModbusCall +1;
		END_IF
	
	32: // wait for FB_Read_Socomec_I61 to be in state 0
		IF FB_Read_Socomec_I61.iStateModbusRead = 0 OR ton_TimeOutState.Q THEN
			i_State_ModbusCall := i_State_ModbusCall + 8;
		END_IF
	
	40:	// next Modbus Poll Call
		FB_Read_Socomec_I61.m_Start := TRUE;
		FB_Read_Socomec_I61.byte_slaveID := 27;
		FB_Read_Socomec_I61.w_Adress := 20490;
		i_State_ModbusCall := i_State_ModbusCall + 1;
	
	41: // wait for received data
		FB_Read_Socomec_I61.m_Start := FALSE;
		IF FB_Read_Socomec_I61.iStateModbusRead = 30 THEN
			lr_Dosierpumpe_2_Freq	:=		FB_Read_Socomec_I61.lr_Freq_Hz	;	
			lr_Dosierpumpe_2_L1N	:=		FB_Read_Socomec_I61.lr_L1N_V	;	
			lr_Dosierpumpe_2_L2N	:=		FB_Read_Socomec_I61.lr_L2N_V	;	
			lr_Dosierpumpe_2_L3N	:=		FB_Read_Socomec_I61.lr_L3N_V	;	
			lr_Dosierpumpe_2_L1L2	:=		FB_Read_Socomec_I61.lr_L1L2_V	;	
			lr_Dosierpumpe_2_L2L3	:=		FB_Read_Socomec_I61.lr_L2L3_V	;	
			lr_Dosierpumpe_2_L3L1	:=		FB_Read_Socomec_I61.lr_L3L1_V	;	
			lr_Dosierpumpe_2_I1		:=		FB_Read_Socomec_I61.lr_I1_A		;	
			lr_Dosierpumpe_2_I2		:=		FB_Read_Socomec_I61.lr_I2_A		;	
			lr_Dosierpumpe_2_I3		:=		FB_Read_Socomec_I61.lr_I3_A		;	
			lr_Dosierpumpe_2_N		:=		FB_Read_Socomec_I61.lr_N_A		;	
			lr_Dosierpumpe_2_P		:=		FB_Read_Socomec_I61.lr_P_kW		;	
			lr_Dosierpumpe_2_Q		:=		FB_Read_Socomec_I61.lr_Q_kVAr	;	
			lr_Dosierpumpe_2_S		:=		FB_Read_Socomec_I61.lr_S_kVA	;	
			lr_Dosierpumpe_2_PF		:=		FB_Read_Socomec_I61.lr_PF		;		
			
			i_State_ModbusCall := i_State_ModbusCall +1;
		END_IF            
		IF FB_Read_Socomec_I61.iStateModbusError = 300 OR ton_TimeOutState.Q THEN
			i_State_ModbusCall := i_State_ModbusCall +1;
		END_IF
	
	42: // wait for FB_Read_Socomec_I61 to be in state 0
		IF FB_Read_Socomec_I61.iStateModbusRead = 0 OR ton_TimeOutState.Q THEN
			i_State_ModbusCall := i_State_ModbusCall + 8;
		END_IF

	50:	// next Modbus Poll Call		first IO10 call
		FB_Read_Socomec_IO10.m_Start := TRUE;
		FB_Read_Socomec_IO10.byte_slaveID := 28;
		FB_Read_Socomec_IO10.w_Adress := 11520;
		i_State_ModbusCall := i_State_ModbusCall + 1;
	
	51: // wait for received data
		FB_Read_Socomec_IO10.m_Start := FALSE;
		IF FB_Read_Socomec_IO10.iStateModbusRead = 30 THEN
			m_Bitumenfuellpumpe_1 := FB_Read_Socomec_IO10.m_Input_Active;		
				
			i_State_ModbusCall := i_State_ModbusCall +1;
		END_IF            
		IF FB_Read_Socomec_IO10.iStateModbusError = 300 OR ton_TimeOutState.Q THEN
			i_State_ModbusCall := i_State_ModbusCall +1;
		END_IF
	
	52: // wait for FB_Read_Socomec_IO10 to be in state 0
		IF FB_Read_Socomec_IO10.iStateModbusRead = 0 OR ton_TimeOutState.Q THEN
			i_State_ModbusCall := i_State_ModbusCall + 8;
		END_IF
		
	60:	// next Modbus Poll Call
		FB_Read_Socomec_I31.m_Start := TRUE;
		FB_Read_Socomec_I31.byte_slaveID := 23;
		FB_Read_Socomec_I31.w_Adress := 18442;
		i_State_ModbusCall := i_State_ModbusCall + 1;
	
	61: // wait for received data
		FB_Read_Socomec_I31.m_Start := FALSE;
		IF FB_Read_Socomec_I31.iStateModbusRead = 30 THEN
			lr_Bitumentank_1_Freq	:=		FB_Read_Socomec_I31.lr_Freq_Hz	;	
			lr_Bitumentank_1_L1N	:=		FB_Read_Socomec_I31.lr_L1N_V	;	
			lr_Bitumentank_1_L2N	:=		FB_Read_Socomec_I31.lr_L2N_V	;	
			lr_Bitumentank_1_L3N	:=		FB_Read_Socomec_I31.lr_L3N_V	;	
			lr_Bitumentank_1_L1L2	:=		FB_Read_Socomec_I31.lr_L1L2_V	;	
			lr_Bitumentank_1_L2L3	:=		FB_Read_Socomec_I31.lr_L2L3_V	;	
			lr_Bitumentank_1_L3L1	:=		FB_Read_Socomec_I31.lr_L3L1_V	;	
			lr_Bitumentank_1_I1		:=		FB_Read_Socomec_I31.lr_I1_A		;	
			lr_Bitumentank_1_I2		:=		FB_Read_Socomec_I31.lr_I2_A		;	
			lr_Bitumentank_1_I3		:=		FB_Read_Socomec_I31.lr_I3_A		;	
			lr_Bitumentank_1_N		:=		FB_Read_Socomec_I31.lr_N_A		;	
			lr_Bitumentank_1_P		:=		FB_Read_Socomec_I31.lr_P_kW		;	
			lr_Bitumentank_1_Q		:=		FB_Read_Socomec_I31.lr_Q_kVAr	;	
			lr_Bitumentank_1_S		:=		FB_Read_Socomec_I31.lr_S_kVA	;	
			lr_Bitumentank_1_PF		:=		FB_Read_Socomec_I31.lr_PF		;		
			
			i_State_ModbusCall := i_State_ModbusCall +1;
		END_IF            
		IF FB_Read_Socomec_I31.iStateModbusError = 300 OR ton_TimeOutState.Q THEN
			i_State_ModbusCall := i_State_ModbusCall +1;
		END_IF
	
	62: // wait for FB_Read_Socomec_I31 to be in state 0
		IF FB_Read_Socomec_I31.iStateModbusRead = 0 OR ton_TimeOutState.Q THEN
			i_State_ModbusCall := i_State_ModbusCall + 8;
		END_IF
		
	70:	// next Modbus Poll Call
		FB_Read_Socomec_I31.m_Start := TRUE;
		FB_Read_Socomec_I31.byte_slaveID := 24;
		FB_Read_Socomec_I31.w_Adress := 18442;
		i_State_ModbusCall := i_State_ModbusCall + 1;
	
	71: // wait for received data
		FB_Read_Socomec_I31.m_Start := FALSE;
		IF FB_Read_Socomec_I31.iStateModbusRead = 30 THEN
			lr_Bitumentank_2_Freq	:=		FB_Read_Socomec_I31.lr_Freq_Hz	;	
			lr_Bitumentank_2_L1N	:=		FB_Read_Socomec_I31.lr_L1N_V	;	
			lr_Bitumentank_2_L2N	:=		FB_Read_Socomec_I31.lr_L2N_V	;	
			lr_Bitumentank_2_L3N	:=		FB_Read_Socomec_I31.lr_L3N_V	;	
			lr_Bitumentank_2_L1L2	:=		FB_Read_Socomec_I31.lr_L1L2_V	;	
			lr_Bitumentank_2_L2L3	:=		FB_Read_Socomec_I31.lr_L2L3_V	;	
			lr_Bitumentank_2_L3L1	:=		FB_Read_Socomec_I31.lr_L3L1_V	;	
			lr_Bitumentank_2_I1		:=		FB_Read_Socomec_I31.lr_I1_A		;	
			lr_Bitumentank_2_I2		:=		FB_Read_Socomec_I31.lr_I2_A		;	
			lr_Bitumentank_2_I3		:=		FB_Read_Socomec_I31.lr_I3_A		;	
			lr_Bitumentank_2_N		:=		FB_Read_Socomec_I31.lr_N_A		;	
			lr_Bitumentank_2_P		:=		FB_Read_Socomec_I31.lr_P_kW		;	
			lr_Bitumentank_2_Q		:=		FB_Read_Socomec_I31.lr_Q_kVAr	;	
			lr_Bitumentank_2_S		:=		FB_Read_Socomec_I31.lr_S_kVA	;	
			lr_Bitumentank_2_PF		:=		FB_Read_Socomec_I31.lr_PF		;		
			
			i_State_ModbusCall := i_State_ModbusCall +1;
		END_IF            
		IF FB_Read_Socomec_I31.iStateModbusError = 300 OR ton_TimeOutState.Q THEN
			i_State_ModbusCall := i_State_ModbusCall +1;
		END_IF
	
	72: // wait for FB_Read_Socomec_I31 to be in state 0
		IF FB_Read_Socomec_I31.iStateModbusRead = 0 OR ton_TimeOutState.Q THEN
			i_State_ModbusCall := i_State_ModbusCall + 8;
		END_IF
		
	80:	// next Modbus Poll Call
		FB_Read_Socomec_I31.m_Start := TRUE;
		FB_Read_Socomec_I31.byte_slaveID := 25;
		FB_Read_Socomec_I31.w_Adress := 18442;
		i_State_ModbusCall := i_State_ModbusCall + 1;
	
	81: // wait for received data
		FB_Read_Socomec_I31.m_Start := FALSE;
		IF FB_Read_Socomec_I31.iStateModbusRead = 30 THEN
			lr_Bitumentank_3_Freq	:=		FB_Read_Socomec_I31.lr_Freq_Hz	;	
			lr_Bitumentank_3_L1N	:=		FB_Read_Socomec_I31.lr_L1N_V	;	
			lr_Bitumentank_3_L2N	:=		FB_Read_Socomec_I31.lr_L2N_V	;	
			lr_Bitumentank_3_L3N	:=		FB_Read_Socomec_I31.lr_L3N_V	;	
			lr_Bitumentank_3_L1L2	:=		FB_Read_Socomec_I31.lr_L1L2_V	;	
			lr_Bitumentank_3_L2L3	:=		FB_Read_Socomec_I31.lr_L2L3_V	;	
			lr_Bitumentank_3_L3L1	:=		FB_Read_Socomec_I31.lr_L3L1_V	;	
			lr_Bitumentank_3_I1		:=		FB_Read_Socomec_I31.lr_I1_A		;	
			lr_Bitumentank_3_I2		:=		FB_Read_Socomec_I31.lr_I2_A		;	
			lr_Bitumentank_3_I3		:=		FB_Read_Socomec_I31.lr_I3_A		;	
			lr_Bitumentank_3_N		:=		FB_Read_Socomec_I31.lr_N_A		;	
			lr_Bitumentank_3_P		:=		FB_Read_Socomec_I31.lr_P_kW		;	
			lr_Bitumentank_3_Q		:=		FB_Read_Socomec_I31.lr_Q_kVAr	;	
			lr_Bitumentank_3_S		:=		FB_Read_Socomec_I31.lr_S_kVA	;	
			lr_Bitumentank_3_PF		:=		FB_Read_Socomec_I31.lr_PF		;		
			
			i_State_ModbusCall := i_State_ModbusCall +1;
		END_IF            
		IF FB_Read_Socomec_I31.iStateModbusError = 300 OR ton_TimeOutState.Q THEN
			i_State_ModbusCall := i_State_ModbusCall +1;
		END_IF
	
	82: // wait for FB_Read_Socomec_I31 to be in state 0
		IF FB_Read_Socomec_I31.iStateModbusRead = 0 OR ton_TimeOutState.Q THEN
			i_State_ModbusCall := i_State_ModbusCall + 8;
		END_IF
		
	90: 
		i_State_ModbusCall := 0;
		
END_CASE

ton_TimeOutState(	IN:= i_State_ModbusCall = i_State_ModbusCall_old, 
					PT:= T#30S, 
					Q=> , 
					ET=> );

i_State_ModbusCall_old := i_State_ModbusCall; 

IF ton_TimeOutState.Q THEN
//	i_State_ModbusCall := 0;
	int_errorCount := int_errorCount  + 1; 
END_IF


tof_TimeOut_Active(	IN:= ton_TimeOutState.Q, 
					PT:=	T#5S , 
					Q=> m_TimeOutActive, 
					ET=> );
IF tof_TimeOut_Active.Q THEN
	 i_State_ErrorActive := i_State_ModbusCall; 
END_IF


FB_Read_Socomec_I61(
	m_Start:= , 
	str_IPAdress:= str_IP , 
	w_Adress:= , 
	uint_port:= , 
	byte_slaveID:= , 
	m_PollSuccessful=> , 
	lr_Freq_Hz=> , 
	lr_L1N_V=> , 
	lr_L2N_V=> , 
	lr_L3N_V=> , 
	lr_L1L2_V=> , 
	lr_L2L3_V=> , 
	lr_L3L1_V=> , 
	lr_I1_A=> , 
	lr_I2_A=> , 
	lr_I3_A=> , 
	lr_N_A=> , 
	lr_P_kW=> , 
	lr_Q_kVAr=> , 
	lr_S_kVA=> , 
	lr_PF=> , 
	udint_Error_ID=> );
	
FB_Read_Socomec_I31(
	m_Start:= , 
	str_IPAdress:= str_IP , 
	w_Adress:= , 
	uint_port:= , 
	byte_slaveID:= , 
	m_PollSuccessful=> , 
	lr_Freq_Hz=> , 
	lr_L1N_V=> , 
	lr_L2N_V=> , 
	lr_L3N_V=> , 
	lr_L1L2_V=> , 
	lr_L2L3_V=> , 
	lr_L3L1_V=> , 
	lr_I1_A=> , 
	lr_I2_A=> , 
	lr_I3_A=> , 
	lr_N_A=> , 
	lr_P_kW=> , 
	lr_Q_kVAr=> , 
	lr_S_kVA=> , 
	lr_PF=> , 
	udint_Error_ID=> );

FB_Read_Socomec_IO10(
	m_Start:= , 
	str_IPAdress:= str_IP , 
	w_Adress:= , 
	uint_port:= , 
	byte_slaveID:= , 
	m_PollSuccessful=> , 
	m_Input_Active=> , 
	udint_Error_ID=> );	

FB_Read_MB(
	m_Enable:= m_Enable, 
	str_IPAdress:= str_IP,
	w_Adress:= word_Adress, 
	usint_Quantity:= usint_Quantity, 
	byte_slaveID:=byte_slaveID,
	uint_port := ,
	m_PollSuccessful=> , 
	w_Array_Received=> , 
	udint_Error_ID=> );

END_PROGRAM

// ---- FB/FB_Socomec_I31.TcPOU
FUNCTION_BLOCK FB_Socomec_I31
VAR_INPUT PERSISTENT
	m_Start						: BOOL;						//starts one modbus read out
	str_IPAdress				: STRING(15);				//IP Adress of the meter
	w_Adress					: WORD;						//modbus adress
	uint_port					: UINT:=502;				//ModbusPort
	byte_slaveID				: BYTE;						//SlaveID of the meter
END_VAR
VAR_OUTPUT
	m_PollSuccessful			: BOOL;						//Poll succesfull		
	lr_Freq_Hz					: LREAL;
	lr_L1N_V					: LREAL;	
	lr_L2N_V					: LREAL;	
	lr_L3N_V					: LREAL;	
	lr_L1L2_V					: LREAL;	
	lr_L2L3_V					: LREAL;	
	lr_L3L1_V					: LREAL;	
	lr_I1_A						: LREAL;	
	lr_I2_A						: LREAL;	
	lr_I3_A						: LREAL;	
	lr_N_A						: LREAL;	
	lr_P_kW						: LREAL;
	lr_Q_kVAr					: LREAL;
	lr_S_kVA					: LREAL;
	lr_PF						: LREAL;	
	udint_Error_ID				: UDINT;					// ERR ID FB_MBReadRegs
END_VAR
VAR
	w_Array_Received			: ARRAY[1..100] OF WORD;	// received data
	timer_Delay					: TON;						//Timer for Delay between Requests
	timer_TimeOut				: TON;						//Timer for Timeout MB Read
	iStateModbusRead			: INT;						//State machine for read out Data over Modbus RTU
	fbMBRead_FC3				: FB_MBReadRegs  ;		//Modbus Read Function (FC3)
	rtrig_Start					: r_trig;					//positive edge for starting the read out
	iStateModbusError			: INT;						//State machine for error out Data over Modbus TCP/IP	
	FPError_FC_3				: R_TRIG;					//Internal positive Edge
	arrBuffer_FC3				: ARRAY[1..100] OF WORD;		//Buffer with Data from FC3
	timer_Connection_ok			: TON;
	int_Data_Received			: INT;
	m_MBTCPError				: BOOL;
	int_Data_Received_old		: INT;
	timer_Connection_ok_TOF	: TOF;
	fbConvertWordToDword		: FB_CV_WORD_TO_DWORD;			//Convert Word to Dword
	m_Poll_ok: BOOL;
	timer_Wait: Ton;
	int_TimeoutError: INT;
	int_FC3Error: INT;
	x: INT;
	i: INT;
	fbConvertWordToudint		: FB_CV_WORD_TO_UDINT;

END_VAR

(*	{attribute 'hide'}--------------------------------------------------------------------------------------------Limits-------------------------------------------------------------------------------------*)

w_Adress := LIMIT(0,w_Adress,60000);

	
(*--------------------------------------------------------------------------------------------State Machine Read--------------------------------------------------------------------------------------*)

//Timer for Delay
timer_Delay(IN:= , PT:= T#50MS, Q=> , ET=> );

//Timeout Timer is dissabled when the Init Step is aktiv or the function is not enabled
IF iStateModbusRead >1 THEN 
	timer_Timeout.IN := FALSE; 
END_IF
timer_Timeout(IN:= , PT:= T#5S, Q=> , ET=> );

//Enable with Delay that not all sockets have to be created at the same time

rtrig_Start(CLK:= m_Start, Q=> );

CASE iStateModbusRead OF

	0://Init Step 
		timer_Delay.IN := FALSE;
		fbMBRead_FC3.bExecute := FALSE;
		m_Poll_ok:=FALSE;
		int_Data_Received:=0;
		FOR i := 1 TO 100 BY 1 DO
			w_Array_Received[i] := 0;
		END_FOR
		iStateModbusRead := 1;
	1: // wait for rtrig START	
		IF rtrig_Start.Q THEN
			iStateModbusRead := 10;
		END_IF
	
	10://read the required registers
		//Start Read
		fbMBRead_FC3.nQuantity := 50;
		fbMBRead_FC3.nMBAddr := w_Adress;
		fbMBRead_FC3.bExecute := TRUE;
		fbMBRead_FC3.nUnitID := byte_slaveID;
		timer_Timeout.IN := TRUE;
		IF fbMBRead_FC3.bBusy THEN 
			timer_Delay.IN := TRUE; 
		END_IF
		
		//Wait for Delay, copy Data and then next step
		IF NOT fbMBRead_FC3.bBusy AND NOT fbMBRead_FC3.bError AND timer_Delay.Q THEN
			m_Poll_ok:=TRUE;
			int_Data_Received:=int_Data_Received+1;
			m_MBTCPError := FALSE; 
			
			w_Array_Received := arrBuffer_FC3;
			
			
			// convert reveived data
			x:=1;
			fbConvertWordToudint(	wInputValue_1:= w_Array_Received[x], 
									wInputValue_2:= w_Array_Received[x+1], 
									eByteOrderForConvert:= eByteOrder.eBigEndian , 
									udiOutputValue=> );
			lr_Freq_Hz:= UDINT_TO_REAL(fbConvertWordToudint.udiOutputValue)/1000;
			x:=3;
			fbConvertWordToudint(	wInputValue_1:= w_Array_Received[x], 
									wInputValue_2:= w_Array_Received[x+1], 
									eByteOrderForConvert:= eByteOrder.eBigEndian , 
									udiOutputValue=> );
			lr_L1N_V:= UDINT_TO_REAL(fbConvertWordToudint.udiOutputValue)/100;
			x:=5;
			fbConvertWordToudint(	wInputValue_1:= w_Array_Received[x], 
									wInputValue_2:= w_Array_Received[x+1], 
									eByteOrderForConvert:= eByteOrder.eBigEndian , 
									udiOutputValue=> );
			lr_L2N_V:= UDINT_TO_REAL(fbConvertWordToudint.udiOutputValue)/100;
			x:=7;
			fbConvertWordToudint(	wInputValue_1:= w_Array_Received[x], 
									wInputValue_2:= w_Array_Received[x+1], 
									eByteOrderForConvert:= eByteOrder.eBigEndian , 
									udiOutputValue=> );
			lr_L3N_V:= UDINT_TO_REAL(fbConvertWordToudint.udiOutputValue)/100;
			
			x:=11;
			fbConvertWordToudint(	wInputValue_1:= w_Array_Received[x], 
									wInputValue_2:= w_Array_Received[x+1], 
									eByteOrderForConvert:= eByteOrder.eBigEndian , 
									udiOutputValue=> );
			lr_L1L2_V:= UDINT_TO_REAL(fbConvertWordToudint.udiOutputValue)/100;
			x:=13;
			fbConvertWordToudint(	wInputValue_1:= w_Array_Received[x], 
									wInputValue_2:= w_Array_Received[x+1], 
									eByteOrderForConvert:= eByteOrder.eBigEndian , 
									udiOutputValue=> );
			lr_L2L3_V:= UDINT_TO_REAL(fbConvertWordToudint.udiOutputValue)/100;
			x:=15;
			fbConvertWordToudint(	wInputValue_1:= w_Array_Received[x], 
									wInputValue_2:= w_Array_Received[x+1], 
									eByteOrderForConvert:= eByteOrder.eBigEndian , 
									udiOutputValue=> );
			lr_L3L1_V:= UDINT_TO_REAL(fbConvertWordToudint.udiOutputValue)/100;
			
			
			x:=17;
			fbConvertWordToudint(	wInputValue_1:= w_Array_Received[x], 
									wInputValue_2:= w_Array_Received[x+1], 
									eByteOrderForConvert:= eByteOrder.eBigEndian , 
									udiOutputValue=> );
			lr_I1_A:= UDINT_TO_REAL(fbConvertWordToudint.udiOutputValue)/1000;
			x:=19;
			fbConvertWordToudint(	wInputValue_1:= w_Array_Received[x], 
									wInputValue_2:= w_Array_Received[x+1], 
									eByteOrderForConvert:= eByteOrder.eBigEndian , 
									udiOutputValue=> );
			lr_I2_A:= UDINT_TO_REAL(fbConvertWordToudint.udiOutputValue)/1000;
			x:=21;
			fbConvertWordToudint(	wInputValue_1:= w_Array_Received[x], 
									wInputValue_2:= w_Array_Received[x+1], 
									eByteOrderForConvert:= eByteOrder.eBigEndian , 
									udiOutputValue=> );
			lr_I3_A:= UDINT_TO_REAL(fbConvertWordToudint.udiOutputValue)/1000;
			x:=23;
			fbConvertWordToudint(	wInputValue_1:= w_Array_Received[x], 
									wInputValue_2:= w_Array_Received[x+1], 
									eByteOrderForConvert:= eByteOrder.eBigEndian , 
									udiOutputValue=> );
			lr_N_A:= UDINT_TO_REAL(fbConvertWordToudint.udiOutputValue)/1000;
			
			x:=35;
			lr_P_kW := DINT_TO_LREAL(DWORD_TO_DINT(w_Array_Received[x]*65536 + w_Array_Received[x+1]))/1000;
			
			x:=37;
			lr_Q_kVAr := DINT_TO_LREAL(DWORD_TO_DINT(w_Array_Received[x]*65536 + w_Array_Received[x+1]))/1000;
			
			
			x:=43;
			fbConvertWordToudint(	wInputValue_1:= w_Array_Received[x], 
									wInputValue_2:= w_Array_Received[x+1], 
									eByteOrderForConvert:= eByteOrder.eBigEndian , 
									udiOutputValue=> );
			lr_S_kVA:= UDINT_TO_REAL(fbConvertWordToudint.udiOutputValue)/1000;
			
			
			x:=45;
			lr_PF := (REAL_TO_LREAL(WORD_TO_INT(w_Array_Received[x])))/1000;
			
			
			//Go to Next Step
			timer_Timeout.IN := FALSE;
			fbMBRead_FC3.bExecute := FALSE;
			timer_Delay.IN := FALSE;		
			iStateModbusRead := 30;
		END_IF	

		//Error or Timeout
		IF FPError_FC_3.Q THEN 
			iStateModbusError := 300;
			int_FC3Error := int_FC3Error+1;
		ELSIF timer_Timeout.Q THEN  
			timer_Timeout.IN := FALSE; 	
			iStateModbusError := 300;
			int_TimeoutError := int_TimeoutError+1;
		END_IF
		
	
	30://Wait and go to step 1
		//1 because 0 is the Init Step for Read
		timer_Wait.IN := TRUE;
		
		IF timer_Wait.Q = TRUE THEN
			iStateModbusRead := 0;
			timer_Wait.IN :=FALSE;
		END_IF

			
		
		//Error on Master, changes on Inputs or Timeout
		IF timer_Timeout.Q THEN 
			iStateModbusError := 300; 
		END_IF
	
END_CASE

(* wait timer*)

timer_Wait(PT:=T#1S);


(*------------------------------------------------------------------Error and Warning----------------------------------------------------------------------------*)	
 
timer_Connection_ok			(In:=int_Data_Received<>int_Data_Received_old,PT:=T#10S);
timer_Connection_ok_TOF		(In:=NOT(int_Data_Received<>int_Data_Received_old) AND int_Data_Received>3 ,PT:=T#20S);
int_Data_Received_old:=int_Data_Received;
m_PollSuccessful:=NOT timer_Connection_ok.Q AND timer_Connection_ok_TOF.Q ;

(*------------------------------------------------------------------------------------------Modbus TCP Functions---------------------------------------------------------------------------------------------*)

fbMBRead_FC3(	sIPAddr:= str_IPAdress, 
				nTCPPort:= uint_port,
				cbLength:= SIZEOF(arrBuffer_FC3), 
				pDestAddr:= ADR(arrBuffer_FC3), 
				tTimeout:= T#10S,
				nErrId => udint_Error_ID);

FPError_FC_3(CLK:= fbMBRead_FC3.bError, Q=> );		

(*------------------------------------------------------------------------------------------State Machine Error---------------------------------------------------------------------------------------------*)	

CASE iStateModbusError OF
	
	300://Error
		timer_Wait.IN :=TRUE;
		timer_Delay.IN := FALSE;
		fbMBRead_FC3.bExecute := FALSE;
		m_MBTCPError := TRUE; 		
		m_Poll_ok:=FALSE;
		int_Data_Received:=0;
				//Restart from new with the Read out part after an Error
		IF timer_Wait.Q = TRUE THEN
			iStateModbusRead := 0;	
			iStateModbusError := 0;
			timer_Wait.IN :=FALSE;
			timer_Timeout.IN := FALSE;
		END_IF		
							
END_CASE

END_FUNCTION_BLOCK

// ---- POUs/prgComEffIO.TcPOU
PROGRAM prgComEffIO
VAR
	fbCom		: FB_MqttCommunicator_V3;
END_VAR

fbCom(
	bConnect:= TRUE, 
	strAuthKey:=  'EIO08031879806' , 
	sUserName:= 'c61b915f-63be-48af-8126-27ef57e2c9fd', 
	sUserPassword:= '93e14dde-8a90-494b-a54c-813d2a465f98', 
	eSavePositionCertificate:= eSavePositionOnPLC.ePostionC, 
	time_HeartBeat_sec := T#1S,
	bConnected=> , 
	bError=> , 
	hrErrorCode=> , 
	eConnectionState=> , 
	eErrorMessage_Out=> );

END_PROGRAM
